// TIA Portal project "智能立库" (V18)

(* hardware
DEVICE "S71500/ET200MP-Station_1"  S7-1500 station
   slot 0: "Profilschiene_0"  Rack  6ES7 590-1***0-0AA0
   slot 0: "PM 70W 120/230VAC"  PM 70W 120/230VAC  6EP1332-4BA00
   slot 1: "PLC_1"  CPU 1516-3 PN/DP  6ES7 516-3AN02-0AB0  V2.9
      slot 3: "CPU-Display_1"  6ES7591-1BA00-0AA0
      slot 32768: "PROFINET-Schnittstelle_1"  X1
         slot 32769: "Port_1"  X1 P1
         slot 32770: "Port_2"  X1 P2
      slot 33024: "PROFINET 接口_1"  X2
      slot 33280: "DP 接口_1"  X3
      slot 34817: "Virtual CP interface port_1"  Virtual CP interface port  Virtual CP interface port
*)

// ===== PLC "PLC_1"  CPU 1516-3 PN/DP =====

VAR_GLOBAL   // PLC tag table "Standard-Variablentabelle"
   "Tag_1" AT %M1000.0 : Bool;
   "Tag_2" AT %M1000.1 : Bool;
   "Tag_3" AT %QW0 : Int;
   "Tag_4" AT %QW1 : Int;
   "Tag_5" AT %QD0 : DWord;
   "Tag_6" AT %QB4 : Byte;
END_VAR

VAR_GLOBAL   // PLC tag table "通讯"
   "确认数量" AT %M200.0 : Bool;
   "出库模式" AT %M200.1 : Bool;
   "入库模式" AT %M200.2 : Bool;
   "启动" AT %M200.3 : Bool;
   "停止" AT %M200.4 : Bool;
   "灰色出库数量" AT %MW202 : Int;
   "绿色出库数量" AT %MW204 : Int;
   "蓝色出库数量" AT %MW206 : Int;
   "取消" AT %M200.5 : Bool;
   "出库启动" AT %M200.6 : Bool;
   "入库启动" AT %M200.7 : Bool;
   "运行标志位" AT %M208.0 : Bool;
   "停止中" AT %M208.1 : Bool;
END_VAR

VAR_GLOBAL   // PLC tag table "仓库数据"
   "1号仓" AT %MW300 : Int;
   "2号仓" AT %MW302 : Int;
   "3号仓" AT %MW304 : Int;
END_VAR

VAR_GLOBAL   // PLC tag table "输入输出"
   "1号仓取货器右移到达" AT %I0.0 : Bool;
   "1号仓取货器左移到达" AT %I0.1 : Bool;
   "1号仓取货器归位" AT %I0.2 : Bool;
   "1号仓取货器运行中" AT %I0.3 : Bool;
   "1号仓码货龙门运行中" AT %I0.4 : Bool;
   "1号仓货物到达传感器" AT %I0.5 : Bool;
   "1号仓货物进入传感器" AT %I0.6 : Bool;
   "1号仓货物离开传感器" AT %I0.7 : Bool;
   "2号仓取货器右移到达" AT %I1.0 : Bool;
   "2号仓取货器左移到达" AT %I1.1 : Bool;
   "2号仓取货器归位" AT %I1.2 : Bool;
   "2号仓取货器运行中" AT %I1.3 : Bool;
   "2号仓码货龙门运行中" AT %I1.4 : Bool;
   "2号仓货物到达传感器" AT %I1.5 : Bool;
   "2号仓货物进入传感器" AT %I1.6 : Bool;
   "2号仓货物离开传感器" AT %I1.7 : Bool;
   "3号仓取货器右移到达" AT %I2.0 : Bool;
   "3号仓取货器左移到达" AT %I2.1 : Bool;
   "3号仓取货器归位" AT %I2.2 : Bool;
   "3号仓取货器运行中" AT %I2.3 : Bool;
   "3号仓码货龙门运行中" AT %I2.4 : Bool;
   "3号仓货物到达传感器" AT %I2.5 : Bool;
   "3号仓货物进入传感器" AT %I2.6 : Bool;
   "3号仓货物离开传感器" AT %I2.7 : Bool;
   "灰色加工中心入料传感器" AT %I3.0 : Bool;
   "灰色加工中心出料传感器" AT %I3.1 : Bool;
   "灰色货箱到达传感器" AT %I3.2 : Bool;
   "绿色加工中心入料传感器" AT %I3.3 : Bool;
   "绿色货箱到达传感器" AT %I3.4 : Bool;
   "绿色加工中心出料传感器" AT %I3.5 : Bool;
   "蓝色加工中心入料传感器" AT %I3.6 : Bool;
   "蓝色加工中心出料传感器" AT %I3.7 : Bool;
   "蓝色货箱到达传感器" AT %I4.0 : Bool;
   "1号仓传送带末端" AT %Q0.0 : Bool;
   "1号仓出货传送带1" AT %Q0.1 : Bool;
   "1号仓出货传送带2" AT %Q0.2 : Bool;
   "1号仓取货器上升" AT %Q0.3 : Bool;
   "1号仓取货器右移" AT %Q0.4 : Bool;
   "1号仓取货器左移" AT %Q0.5 : Bool;
   "1号仓货物进入传送带" AT %Q0.6 : Bool;
   "1号仓进货传送带" AT %Q0.7 : Bool;
   "2号仓传送带末端" AT %Q1.0 : Bool;
   "2号仓出货传送带1" AT %Q1.1 : Bool;
   "2号仓出货传送带2" AT %Q1.2 : Bool;
   "2号仓取货器上升" AT %Q1.3 : Bool;
   "2号仓取货器右移" AT %Q1.4 : Bool;
   "2号仓取货器左移" AT %Q1.5 : Bool;
   "2号仓货物进入传送带" AT %Q1.6 : Bool;
   "2号仓进货传送带" AT %Q1.7 : Bool;
   "3号仓传送带末端" AT %Q2.0 : Bool;
   "3号仓出货传送带1" AT %Q2.1 : Bool;
   "3号仓出货传送带2" AT %Q2.2 : Bool;
   "3号仓取货器上升" AT %Q2.3 : Bool;
   "3号仓取货器右移" AT %Q2.4 : Bool;
   "3号仓取货器左移" AT %Q2.5 : Bool;
   "3号仓货物进入传送带" AT %Q2.6 : Bool;
   "3号仓进货传送带" AT %Q2.7 : Bool;
   "灰色加工中心停止" AT %Q3.0 : Bool;
   "灰色加工中心入料传送带" AT %Q3.1 : Bool;
   "灰色加工中心出料传送带1" AT %Q3.2 : Bool;
   "灰色加工中心出料传送带2" AT %Q3.3 : Bool;
   "灰色加工中心加工上盖使能" AT %Q3.4 : Bool;
   "灰色加工中心启动" AT %Q3.5 : Bool;
   "绿色加工中心停止" AT %Q3.6 : Bool;
   "绿色加工中心入料传送带" AT %Q3.7 : Bool;
   "绿色加工中心出料传送带1" AT %Q4.0 : Bool;
   "绿色加工中心出料传送带2" AT %Q4.1 : Bool;
   "绿色加工中心加工上盖使能" AT %Q4.2 : Bool;
   "绿色加工中心启动" AT %Q4.3 : Bool;
   "蓝色加工中心停止" AT %Q4.4 : Bool;
   "蓝色加工中心入料传送带" AT %Q4.5 : Bool;
   "蓝色加工中心出料传送带1" AT %Q4.6 : Bool;
   "蓝色加工中心出料传送带2" AT %Q4.7 : Bool;
   "蓝色加工中心加工上盖使能" AT %Q5.0 : Bool;
   "蓝色加工中心启动" AT %Q5.1 : Bool;
   "1号仓目标仓位" AT %QD48 : DInt;
   "2号仓目标仓位" AT %QD52 : DInt;
   "3号仓目标仓位" AT %QD56 : DInt;
END_VAR

DATA_BLOCK "模式切换"   // DB1
{ S7_Optimized_Access := 'TRUE' }
VERSION : 0.1
   VAR
      出库模式 : Struct
         中间 : Bool;
         启动 : Bool;
         确认数量 : Bool;
         全部出库完成 : Bool;
      END_STRUCT;
      入库模式 : Struct
         中间 : Bool;
         启动 : Bool;
         入库完成保持 : Struct
            "1" : Bool;
            "2" : Bool;
            "3" : Bool;
            汇总 : Bool;
         END_STRUCT;
      END_STRUCT;
      沿 : Struct
         "1" : Bool;
         "2" : Bool;
         "3" : Bool;
         "4" : Bool;
         "5" : Bool;
      END_STRUCT;
   END_VAR
BEGIN
END_DATA_BLOCK

DATA_BLOCK "2号仓库汇总块_DB"   // DB2
{ S7_Optimized_Access := 'TRUE' }
VERSION : 0.1
// stored: InstanceOfName 汇总块
"汇总块"
BEGIN
END_DATA_BLOCK

DATA_BLOCK "3号仓库汇总块_DB"   // DB3
{ S7_Optimized_Access := 'TRUE' }
VERSION : 0.1
// stored: InstanceOfName 汇总块
"汇总块"
BEGIN
END_DATA_BLOCK

DATA_BLOCK "手动调试模式数据"   // DB4
{ S7_Optimized_Access := 'FALSE' }
VERSION : 0.1
   VAR
      传感器数据 : Struct
         "1号仓取货器右移到达" : Bool;
         "1号仓取货器左移到达" : Bool;
         "1号仓取货器归位" : Bool;
         "1号仓取货器运行中" : Bool;
         "1号仓码货龙门运行中" : Bool;
         "1号仓货物到达传感器" : Bool;
         "1号仓货物进入传感器" : Bool;
         "1号仓货物离开传感器" : Bool;
         "2号仓取货器右移到达" : Bool;
         "2号仓取货器左移到达" : Bool;
         "2号仓取货器归位" : Bool;
         "2号仓取货器运行中" : Bool;
         "2号仓码货龙门运行中" : Bool;
         "2号仓货物到达传感器" : Bool;
         "2号仓货物进入传感器" : Bool;
         "2号仓货物离开传感器" : Bool;
         "3号仓取货器右移到达" : Bool;
         "3号仓取货器左移到达" : Bool;
         "3号仓取货器归位" : Bool;
         "3号仓取货器运行中" : Bool;
         "3号仓码货龙门运行中" : Bool;
         "3号仓货物到达传感器" : Bool;
         "3号仓货物进入传感器" : Bool;
         "3号仓货物离开传感器" : Bool;
         灰色加工中心入料传感器 : Bool;
         灰色加工中心出料传感器 : Bool;
         灰色货箱到达传感器 : Bool;
         绿色加工中心入料传感器 : Bool;
         绿色货箱到达传感器 : Bool;
         绿色加工中心出料传感器 : Bool;
         蓝色加工中心入料传感器 : Bool;
         蓝色加工中心出料传感器 : Bool;
         蓝色货箱到达传感器 : Bool;
      END_STRUCT;
      执行器 : Struct
         "1号仓传送带末端" : Bool;
         "1号仓出货传送带1" : Bool;
         "1号仓出货传送带2" : Bool;
         "1号仓取货器上升" : Bool;
         "1号仓取货器右移" : Bool;
         "1号仓取货器左移" : Bool;
         "1号仓货物进入传送带" : Bool;
         "1号仓进货传送带" : Bool;
         "2号仓传送带末端" : Bool;
         "2号仓出货传送带1" : Bool;
         "2号仓出货传送带2" : Bool;
         "2号仓取货器上升" : Bool;
         "2号仓取货器右移" : Bool;
         "2号仓取货器左移" : Bool;
         "2号仓货物进入传送带" : Bool;
         "2号仓进货传送带" : Bool;
         "3号仓传送带末端" : Bool;
         "3号仓出货传送带1" : Bool;
         "3号仓出货传送带2" : Bool;
         "3号仓取货器上升" : Bool;
         "3号仓取货器右移" : Bool;
         "3号仓取货器左移" : Bool;
         "3号仓货物进入传送带" : Bool;
         "3号仓进货传送带" : Bool;
         灰色加工中心停止 : Bool;
         灰色加工中心入料传送带 : Bool;
         灰色加工中心出料传送带1 : Bool;
         灰色加工中心出料传送带2 : Bool;
         灰色加工中心加工上盖使能 : Bool;
         灰色加工中心启动 : Bool;
         绿色加工中心停止 : Bool;
         绿色加工中心入料传送带 : Bool;
         绿色加工中心出料传送带1 : Bool;
         绿色加工中心出料传送带2 : Bool;
         绿色加工中心加工上盖使能 : Bool;
         绿色加工中心启动 : Bool;
         蓝色加工中心停止 : Bool;
         蓝色加工中心入料传送带 : Bool;
         蓝色加工中心出料传送带1 : Bool;
         蓝色加工中心出料传送带2 : Bool;
         蓝色加工中心加工上盖使能 : Bool;
         蓝色加工中心启动 : Bool;
      END_STRUCT;
   END_VAR
BEGIN
END_DATA_BLOCK

DATA_BLOCK "1号仓库汇总块_DB"   // DB7
{ S7_Optimized_Access := 'TRUE' }
VERSION : 0.1
// stored: InstanceOfName 汇总块
"汇总块"
BEGIN
END_DATA_BLOCK

FUNCTION_BLOCK "取货器"   // FB1, LAD
{ S7_Optimized_Access := 'TRUE' }
VERSION : 0.1
   VAR_INPUT
      传送带进货 : Bool;
      "传送带出货/仓库进货" : Bool;
      仓库出货 : Bool;
      取货器左移到达 : Bool;
      取货器右移到达 : Bool;
      取货器归位 : Bool;
      取货器运行中 : Bool;
   END_VAR
   VAR_OUTPUT
      取货臂左移 : Bool;
      取货臂右移 : Bool;
      取货器上升 : Bool;
      传送带进货完成 : Bool;
      "传送带出货/仓库进货完成" : Bool;
      仓库出货完成 : Bool;
   END_VAR
   VAR
      传送带进货运行步 : Int;
      传送带出货运行步 : Int;
      仓库出货运行步 : Int;
      传送带进货沿缓冲位 : Struct
         "1" : Bool;
         "2" : Bool;
         "3" : Bool;
         "4" : Bool;
         "5" : Bool;
         "6" : Bool;
      END_STRUCT;
      "传送带出货/仓库进货沿缓冲位" : Struct
         "1" : Bool;
         "2" : Bool;
         "3" : Bool;
         "4" : Bool;
         "5" : Bool;
      END_STRUCT;
      仓库出货沿缓冲位 : Struct
         "1" : Bool;
         "2" : Bool;
         "3" : Bool;
         "4" : Bool;
         "5" : Bool;
      END_STRUCT;
   END_VAR
   VAR_TEMP   // added for the SCL form of the ladder/FBD networks
      _w1 : Bool;
      _w2 : Bool;
      _w3 : Bool;
      _w4 : Bool;
      _w5 : Bool;
      _w6 : Bool;
      _w7 : Bool;
      _w8 : Bool;
      _w9 : Bool;
   END_VAR
BEGIN

REGION Network 1: 传送带进货
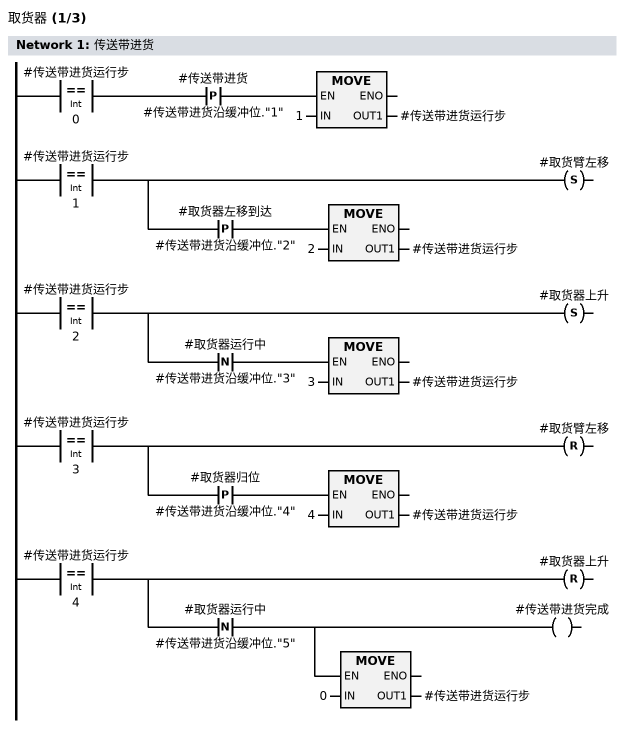
   RUNG wire#powerrail
      { S7_Templates := "SrcType := Int" } EQ_Contact(in1 := #传送带进货运行步, in2 := 0)
      P_Contact(operand := #传送带进货, bit := #传送带进货沿缓冲位."1")
      Move(in := 1, out1 => #传送带进货运行步)
   END_RUNG
   RUNG wire#powerrail
      { S7_Templates := "SrcType := Int" } EQ_Contact(in1 := #传送带进货运行步, in2 := 1)
      wire#w1
      S_Coil( #取货臂左移 )
   END_RUNG
   RUNG wire#w1
      P_Contact(operand := #取货器左移到达, bit := #传送带进货沿缓冲位."2")
      Move(in := 2, out1 => #传送带进货运行步)
   END_RUNG
   RUNG wire#powerrail
      { S7_Templates := "SrcType := Int" } EQ_Contact(in1 := #传送带进货运行步, in2 := 2)
      wire#w2
      S_Coil( #取货器上升 )
   END_RUNG
   RUNG wire#w2
      N_Contact(operand := #取货器运行中, bit := #传送带进货沿缓冲位."3")
      Move(in := 3, out1 => #传送带进货运行步)
   END_RUNG
   RUNG wire#powerrail
      { S7_Templates := "SrcType := Int" } EQ_Contact(in1 := #传送带进货运行步, in2 := 3)
      wire#w3
      R_Coil( #取货臂左移 )
   END_RUNG
   RUNG wire#w3
      P_Contact(operand := #取货器归位, bit := #传送带进货沿缓冲位."4")
      Move(in := 4, out1 => #传送带进货运行步)
   END_RUNG
   RUNG wire#powerrail
      { S7_Templates := "SrcType := Int" } EQ_Contact(in1 := #传送带进货运行步, in2 := 4)
      wire#w4
      R_Coil( #取货器上升 )
   END_RUNG
   RUNG wire#w4
      N_Contact(operand := #取货器运行中, bit := #传送带进货沿缓冲位."5")
      wire#w5
      Coil( #传送带进货完成 )
   END_RUNG
   RUNG wire#w5
      Move(in := 0, out1 => #传送带进货运行步)
   END_RUNG
   // the same network as SCL:
   #_w1 := (#传送带进货运行步 = 0) AND #传送带进货 AND NOT #传送带进货沿缓冲位."1";   // rising edge of #传送带进货
   #传送带进货沿缓冲位."1" := #传送带进货;
   IF #_w1 THEN #传送带进货运行步 := 1; END_IF;
   #_w2 := #传送带进货运行步 = 1;
   IF #_w2 THEN #取货臂左移 := TRUE; END_IF;
   #_w3 := #_w2 AND #取货器左移到达 AND NOT #传送带进货沿缓冲位."2";   // rising edge of #取货器左移到达
   #传送带进货沿缓冲位."2" := #取货器左移到达;
   IF #_w3 THEN #传送带进货运行步 := 2; END_IF;
   #_w4 := #传送带进货运行步 = 2;
   IF #_w4 THEN #取货器上升 := TRUE; END_IF;
   #_w5 := #_w4 AND NOT #取货器运行中 AND #传送带进货沿缓冲位."3";   // falling edge of #取货器运行中
   #传送带进货沿缓冲位."3" := #取货器运行中;
   IF #_w5 THEN #传送带进货运行步 := 3; END_IF;
   #_w6 := #传送带进货运行步 = 3;
   IF #_w6 THEN #取货臂左移 := FALSE; END_IF;
   #_w7 := #_w6 AND #取货器归位 AND NOT #传送带进货沿缓冲位."4";   // rising edge of #取货器归位
   #传送带进货沿缓冲位."4" := #取货器归位;
   IF #_w7 THEN #传送带进货运行步 := 4; END_IF;
   #_w8 := #传送带进货运行步 = 4;
   IF #_w8 THEN #取货器上升 := FALSE; END_IF;
   #_w9 := #_w8 AND NOT #取货器运行中 AND #传送带进货沿缓冲位."5";   // falling edge of #取货器运行中
   #传送带进货沿缓冲位."5" := #取货器运行中;
   #传送带进货完成 := #_w9;
   IF #_w9 THEN #传送带进货运行步 := 0; END_IF;
END_REGION

REGION Network 2: 传送带出货/仓库进货
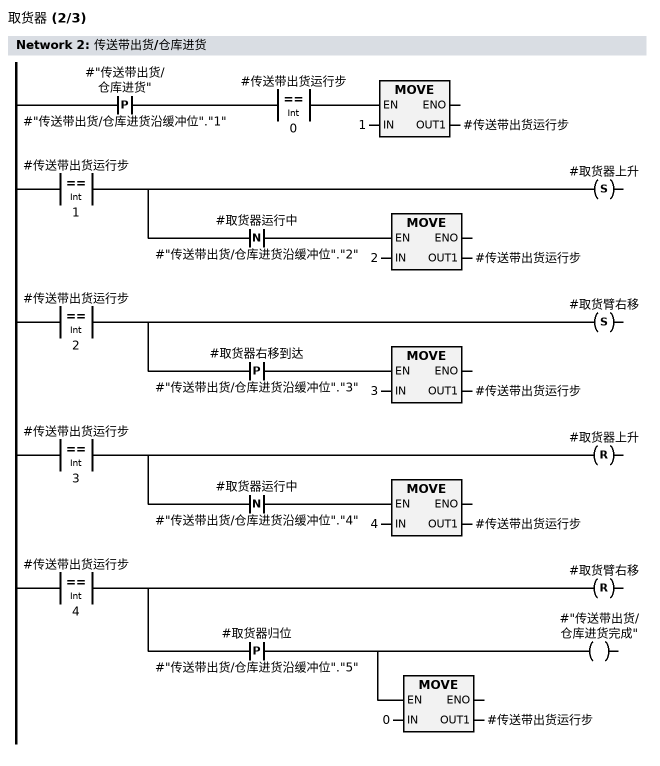
   RUNG wire#powerrail
      P_Contact(operand := #"传送带出货/仓库进货", bit := #"传送带出货/仓库进货沿缓冲位"."1")
      { S7_Templates := "SrcType := Int" } EQ_Contact(in1 := #传送带出货运行步, in2 := 0)
      Move(in := 1, out1 => #传送带出货运行步)
   END_RUNG
   RUNG wire#powerrail
      { S7_Templates := "SrcType := Int" } EQ_Contact(in1 := #传送带出货运行步, in2 := 1)
      wire#w1
      S_Coil( #取货器上升 )
   END_RUNG
   RUNG wire#w1
      N_Contact(operand := #取货器运行中, bit := #"传送带出货/仓库进货沿缓冲位"."2")
      Move(in := 2, out1 => #传送带出货运行步)
   END_RUNG
   RUNG wire#powerrail
      { S7_Templates := "SrcType := Int" } EQ_Contact(in1 := #传送带出货运行步, in2 := 2)
      wire#w2
      S_Coil( #取货臂右移 )
   END_RUNG
   RUNG wire#w2
      P_Contact(operand := #取货器右移到达, bit := #"传送带出货/仓库进货沿缓冲位"."3")
      Move(in := 3, out1 => #传送带出货运行步)
   END_RUNG
   RUNG wire#powerrail
      { S7_Templates := "SrcType := Int" } EQ_Contact(in1 := #传送带出货运行步, in2 := 3)
      wire#w3
      R_Coil( #取货器上升 )
   END_RUNG
   RUNG wire#w3
      N_Contact(operand := #取货器运行中, bit := #"传送带出货/仓库进货沿缓冲位"."4")
      Move(in := 4, out1 => #传送带出货运行步)
   END_RUNG
   RUNG wire#powerrail
      { S7_Templates := "SrcType := Int" } EQ_Contact(in1 := #传送带出货运行步, in2 := 4)
      wire#w4
      R_Coil( #取货臂右移 )
   END_RUNG
   RUNG wire#w4
      P_Contact(operand := #取货器归位, bit := #"传送带出货/仓库进货沿缓冲位"."5")
      wire#w5
      Coil( #"传送带出货/仓库进货完成" )
   END_RUNG
   RUNG wire#w5
      Move(in := 0, out1 => #传送带出货运行步)
   END_RUNG
   // the same network as SCL:
   #_w1 := #"传送带出货/仓库进货" AND NOT #"传送带出货/仓库进货沿缓冲位"."1";   // rising edge of #"传送带出货/仓库进货"
   #"传送带出货/仓库进货沿缓冲位"."1" := #"传送带出货/仓库进货";
   IF #_w1 AND (#传送带出货运行步 = 0) THEN #传送带出货运行步 := 1; END_IF;
   #_w2 := #传送带出货运行步 = 1;
   IF #_w2 THEN #取货器上升 := TRUE; END_IF;
   #_w3 := #_w2 AND NOT #取货器运行中 AND #"传送带出货/仓库进货沿缓冲位"."2";   // falling edge of #取货器运行中
   #"传送带出货/仓库进货沿缓冲位"."2" := #取货器运行中;
   IF #_w3 THEN #传送带出货运行步 := 2; END_IF;
   #_w4 := #传送带出货运行步 = 2;
   IF #_w4 THEN #取货臂右移 := TRUE; END_IF;
   #_w5 := #_w4 AND #取货器右移到达 AND NOT #"传送带出货/仓库进货沿缓冲位"."3";   // rising edge of #取货器右移到达
   #"传送带出货/仓库进货沿缓冲位"."3" := #取货器右移到达;
   IF #_w5 THEN #传送带出货运行步 := 3; END_IF;
   #_w6 := #传送带出货运行步 = 3;
   IF #_w6 THEN #取货器上升 := FALSE; END_IF;
   #_w7 := #_w6 AND NOT #取货器运行中 AND #"传送带出货/仓库进货沿缓冲位"."4";   // falling edge of #取货器运行中
   #"传送带出货/仓库进货沿缓冲位"."4" := #取货器运行中;
   IF #_w7 THEN #传送带出货运行步 := 4; END_IF;
   #_w8 := #传送带出货运行步 = 4;
   IF #_w8 THEN #取货臂右移 := FALSE; END_IF;
   #_w9 := #_w8 AND #取货器归位 AND NOT #"传送带出货/仓库进货沿缓冲位"."5";   // rising edge of #取货器归位
   #"传送带出货/仓库进货沿缓冲位"."5" := #取货器归位;
   #"传送带出货/仓库进货完成" := #_w9;
   IF #_w9 THEN #传送带出货运行步 := 0; END_IF;
END_REGION

REGION Network 3: 仓库出货
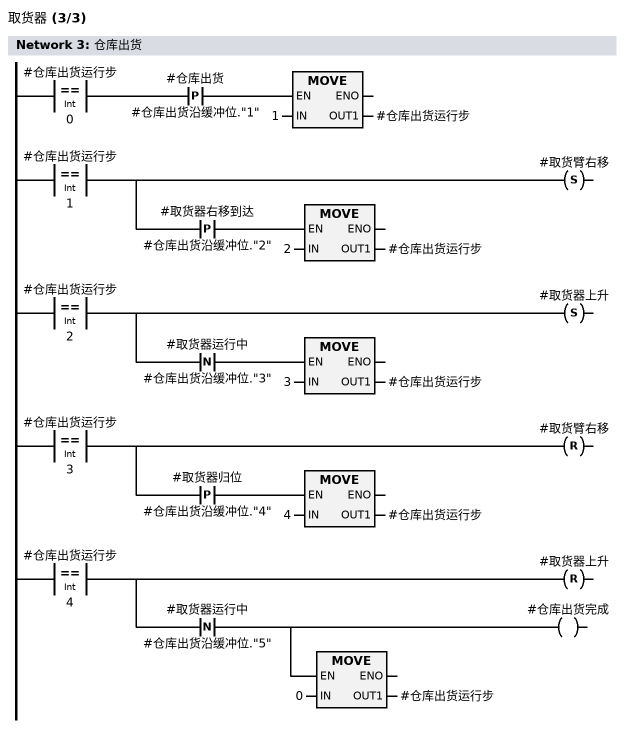
   RUNG wire#powerrail
      { S7_Templates := "SrcType := Int" } EQ_Contact(in1 := #仓库出货运行步, in2 := 0)
      P_Contact(operand := #仓库出货, bit := #仓库出货沿缓冲位."1")
      Move(in := 1, out1 => #仓库出货运行步)
   END_RUNG
   RUNG wire#powerrail
      { S7_Templates := "SrcType := Int" } EQ_Contact(in1 := #仓库出货运行步, in2 := 1)
      wire#w1
      S_Coil( #取货臂右移 )
   END_RUNG
   RUNG wire#w1
      P_Contact(operand := #取货器右移到达, bit := #仓库出货沿缓冲位."2")
      Move(in := 2, out1 => #仓库出货运行步)
   END_RUNG
   RUNG wire#powerrail
      { S7_Templates := "SrcType := Int" } EQ_Contact(in1 := #仓库出货运行步, in2 := 2)
      wire#w2
      S_Coil( #取货器上升 )
   END_RUNG
   RUNG wire#w2
      N_Contact(operand := #取货器运行中, bit := #仓库出货沿缓冲位."3")
      Move(in := 3, out1 => #仓库出货运行步)
   END_RUNG
   RUNG wire#powerrail
      { S7_Templates := "SrcType := Int" } EQ_Contact(in1 := #仓库出货运行步, in2 := 3)
      wire#w3
      R_Coil( #取货臂右移 )
   END_RUNG
   RUNG wire#w3
      P_Contact(operand := #取货器归位, bit := #仓库出货沿缓冲位."4")
      Move(in := 4, out1 => #仓库出货运行步)
   END_RUNG
   RUNG wire#powerrail
      { S7_Templates := "SrcType := Int" } EQ_Contact(in1 := #仓库出货运行步, in2 := 4)
      wire#w4
      R_Coil( #取货器上升 )
   END_RUNG
   RUNG wire#w4
      N_Contact(operand := #取货器运行中, bit := #仓库出货沿缓冲位."5")
      wire#w5
      Coil( #仓库出货完成 )
   END_RUNG
   RUNG wire#w5
      Move(in := 0, out1 => #仓库出货运行步)
   END_RUNG
   // the same network as SCL:
   #_w1 := (#仓库出货运行步 = 0) AND #仓库出货 AND NOT #仓库出货沿缓冲位."1";   // rising edge of #仓库出货
   #仓库出货沿缓冲位."1" := #仓库出货;
   IF #_w1 THEN #仓库出货运行步 := 1; END_IF;
   #_w2 := #仓库出货运行步 = 1;
   IF #_w2 THEN #取货臂右移 := TRUE; END_IF;
   #_w3 := #_w2 AND #取货器右移到达 AND NOT #仓库出货沿缓冲位."2";   // rising edge of #取货器右移到达
   #仓库出货沿缓冲位."2" := #取货器右移到达;
   IF #_w3 THEN #仓库出货运行步 := 2; END_IF;
   #_w4 := #仓库出货运行步 = 2;
   IF #_w4 THEN #取货器上升 := TRUE; END_IF;
   #_w5 := #_w4 AND NOT #取货器运行中 AND #仓库出货沿缓冲位."3";   // falling edge of #取货器运行中
   #仓库出货沿缓冲位."3" := #取货器运行中;
   IF #_w5 THEN #仓库出货运行步 := 3; END_IF;
   #_w6 := #仓库出货运行步 = 3;
   IF #_w6 THEN #取货臂右移 := FALSE; END_IF;
   #_w7 := #_w6 AND #取货器归位 AND NOT #仓库出货沿缓冲位."4";   // rising edge of #取货器归位
   #仓库出货沿缓冲位."4" := #取货器归位;
   IF #_w7 THEN #仓库出货运行步 := 4; END_IF;
   #_w8 := #仓库出货运行步 = 4;
   IF #_w8 THEN #取货器上升 := FALSE; END_IF;
   #_w9 := #_w8 AND NOT #取货器运行中 AND #仓库出货沿缓冲位."5";   // falling edge of #取货器运行中
   #仓库出货沿缓冲位."5" := #取货器运行中;
   #仓库出货完成 := #_w9;
   IF #_w9 THEN #仓库出货运行步 := 0; END_IF;
END_REGION
END_FUNCTION_BLOCK

FUNCTION_BLOCK "龙门码货机"   // FB2, LAD
{ S7_Optimized_Access := 'TRUE' }
VERSION : 0.1
   VAR_INPUT
      仓位号输入 : Int;
      入库 : Bool;
      出库 : Bool;
      龙门运行中 : Bool;
      取货器左移到达传感器 : Bool;
      取货器右移到达传感器 : Bool;
      取货器归位传感器 : Bool;
      取货器运行传感器 : Bool;
   END_VAR
   VAR_OUTPUT
      仓位号输出 : DInt;
      取货臂左移 : Bool;
      取货臂右移 : Bool;
      取货器上升 : Bool;
      入库完成 : Bool;
      出库完成 : Bool;
   END_VAR
   VAR
      入库步骤号 : Int;
      出库步骤号 : Int;
      入库沿缓冲位 : Struct
         "1" : Bool;
         "2" : Bool;
         "3" : Bool;
         "4" : Bool;
      END_STRUCT;
      出库沿缓冲位 : Struct
         "1" : Bool;
         "2" : Bool;
         "3" : Bool;
         "4" : Bool;
      END_STRUCT;
      取货器_Instance : "取货器";
   END_VAR
   VAR_TEMP   // added for the SCL form of the ladder/FBD networks
      _w1 : Bool;
      _w2 : Bool;
      _w3 : Bool;
      _w4 : Bool;
      _w5 : Bool;
      _w6 : Bool;
      _w7 : Bool;
      _w8 : Bool;
      _w9 : Bool;
   END_VAR
BEGIN

REGION Network 1: 入库
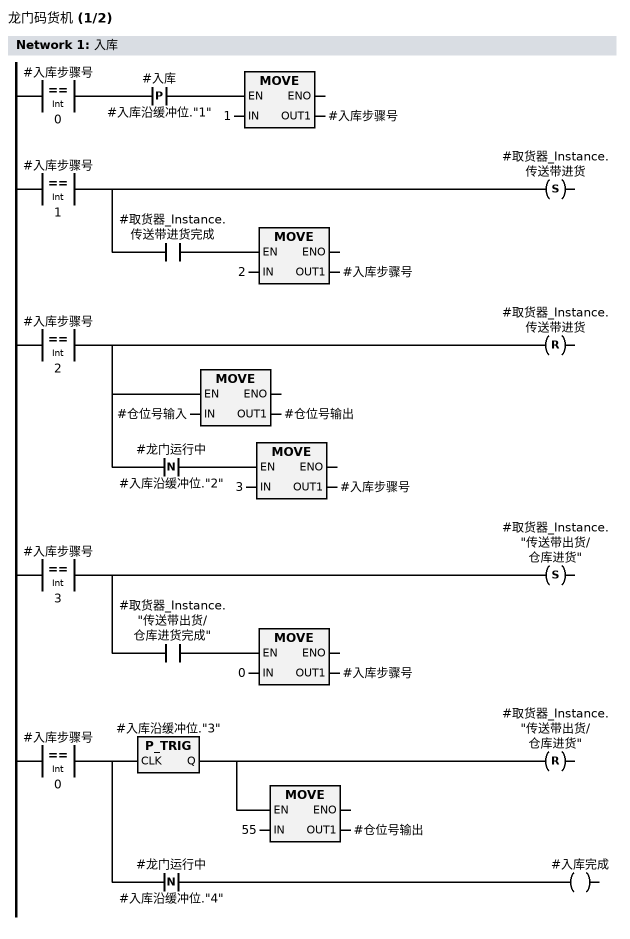
   RUNG wire#powerrail
      { S7_Templates := "SrcType := Int" } EQ_Contact(in1 := #入库步骤号, in2 := 0)
      P_Contact(operand := #入库, bit := #入库沿缓冲位."1")
      Move(in := 1, out1 => #入库步骤号)
   END_RUNG
   RUNG wire#powerrail
      { S7_Templates := "SrcType := Int" } EQ_Contact(in1 := #入库步骤号, in2 := 1)
      wire#w1
      S_Coil( #取货器_Instance.传送带进货 )
   END_RUNG
   RUNG wire#w1
      Contact( #取货器_Instance.传送带进货完成 )
      Move(in := 2, out1 => #入库步骤号)
   END_RUNG
   RUNG wire#powerrail
      { S7_Templates := "SrcType := Int" } EQ_Contact(in1 := #入库步骤号, in2 := 2)
      wire#w2
      R_Coil( #取货器_Instance.传送带进货 )
   END_RUNG
   RUNG wire#w2
      Move(in := #仓位号输入, out1 => #仓位号输出)
   END_RUNG
   RUNG wire#w2
      N_Contact(operand := #龙门运行中, bit := #入库沿缓冲位."2")
      Move(in := 3, out1 => #入库步骤号)
   END_RUNG
   RUNG wire#powerrail
      { S7_Templates := "SrcType := Int" } EQ_Contact(in1 := #入库步骤号, in2 := 3)
      wire#w3
      S_Coil( #取货器_Instance."传送带出货/仓库进货" )
   END_RUNG
   RUNG wire#w3
      Contact( #取货器_Instance."传送带出货/仓库进货完成" )
      Move(in := 0, out1 => #入库步骤号)
   END_RUNG
   RUNG wire#powerrail
      { S7_Templates := "SrcType := Int" } EQ_Contact(in1 := #入库步骤号, in2 := 0)
      wire#w4
      P_Trig( #入库沿缓冲位."3" )
      wire#w5
      R_Coil( #取货器_Instance."传送带出货/仓库进货" )
   END_RUNG
   RUNG wire#w5
      Move(in := 55, out1 => #仓位号输出)
   END_RUNG
   RUNG wire#w4
      N_Contact(operand := #龙门运行中, bit := #入库沿缓冲位."4")
      Coil( #入库完成 )
   END_RUNG
   // the same network as SCL:
   #_w1 := (#入库步骤号 = 0) AND #入库 AND NOT #入库沿缓冲位."1";   // rising edge of #入库
   #入库沿缓冲位."1" := #入库;
   IF #_w1 THEN #入库步骤号 := 1; END_IF;
   #_w2 := #入库步骤号 = 1;
   IF #_w2 THEN #取货器_Instance.传送带进货 := TRUE; END_IF;
   IF #_w2 AND #取货器_Instance.传送带进货完成 THEN #入库步骤号 := 2; END_IF;
   #_w3 := #入库步骤号 = 2;
   IF #_w3 THEN
       #取货器_Instance.传送带进货 := FALSE;
       #仓位号输出 := #仓位号输入;
   END_IF;
   #_w4 := #_w3 AND NOT #龙门运行中 AND #入库沿缓冲位."2";   // falling edge of #龙门运行中
   #入库沿缓冲位."2" := #龙门运行中;
   IF #_w4 THEN #入库步骤号 := 3; END_IF;
   #_w5 := #入库步骤号 = 3;
   IF #_w5 THEN #取货器_Instance."传送带出货/仓库进货" := TRUE; END_IF;
   IF #_w5 AND #取货器_Instance."传送带出货/仓库进货完成" THEN #入库步骤号 := 0; END_IF;
   #_w6 := #入库步骤号 = 0;
   #_w7 := #_w6 AND NOT #入库沿缓冲位."3";   // rising edge
   #入库沿缓冲位."3" := #_w6;
   IF #_w7 THEN
       #取货器_Instance."传送带出货/仓库进货" := FALSE;
       #仓位号输出 := 55;
   END_IF;
   #_w8 := #_w6 AND NOT #龙门运行中 AND #入库沿缓冲位."4";   // falling edge of #龙门运行中
   #入库沿缓冲位."4" := #龙门运行中;
   #入库完成 := #_w8;
END_REGION

REGION Network 2: 出库
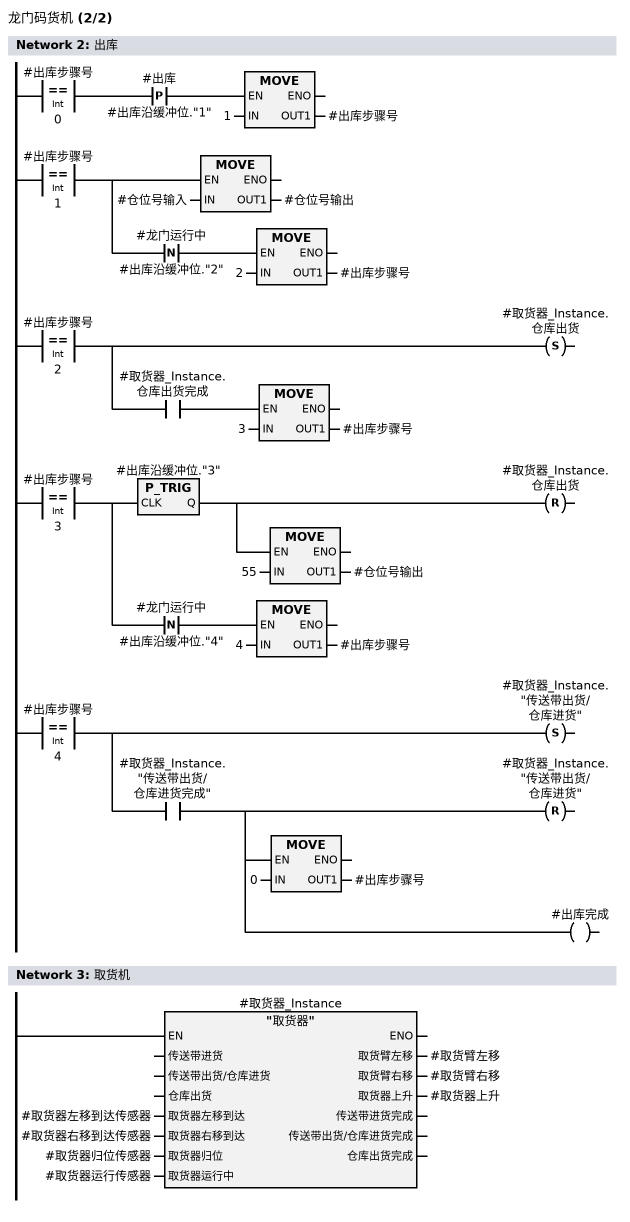
   RUNG wire#powerrail
      { S7_Templates := "SrcType := Int" } EQ_Contact(in1 := #出库步骤号, in2 := 0)
      P_Contact(operand := #出库, bit := #出库沿缓冲位."1")
      Move(in := 1, out1 => #出库步骤号)
   END_RUNG
   RUNG wire#powerrail
      { S7_Templates := "SrcType := Int" } EQ_Contact(in1 := #出库步骤号, in2 := 1)
      wire#w1
      Move(in := #仓位号输入, out1 => #仓位号输出)
   END_RUNG
   RUNG wire#w1
      N_Contact(operand := #龙门运行中, bit := #出库沿缓冲位."2")
      Move(in := 2, out1 => #出库步骤号)
   END_RUNG
   RUNG wire#powerrail
      { S7_Templates := "SrcType := Int" } EQ_Contact(in1 := #出库步骤号, in2 := 2)
      wire#w2
      S_Coil( #取货器_Instance.仓库出货 )
   END_RUNG
   RUNG wire#w2
      Contact( #取货器_Instance.仓库出货完成 )
      Move(in := 3, out1 => #出库步骤号)
   END_RUNG
   RUNG wire#powerrail
      { S7_Templates := "SrcType := Int" } EQ_Contact(in1 := #出库步骤号, in2 := 3)
      wire#w3
      P_Trig( #出库沿缓冲位."3" )
      wire#w4
      R_Coil( #取货器_Instance.仓库出货 )
   END_RUNG
   RUNG wire#w4
      Move(in := 55, out1 => #仓位号输出)
   END_RUNG
   RUNG wire#w3
      N_Contact(operand := #龙门运行中, bit := #出库沿缓冲位."4")
      Move(in := 4, out1 => #出库步骤号)
   END_RUNG
   RUNG wire#powerrail
      { S7_Templates := "SrcType := Int" } EQ_Contact(in1 := #出库步骤号, in2 := 4)
      wire#w5
      S_Coil( #取货器_Instance."传送带出货/仓库进货" )
   END_RUNG
   RUNG wire#w5
      Contact( #取货器_Instance."传送带出货/仓库进货完成" )
      wire#w6
      R_Coil( #取货器_Instance."传送带出货/仓库进货" )
   END_RUNG
   RUNG wire#w6
      Move(in := 0, out1 => #出库步骤号)
   END_RUNG
   RUNG wire#w6
      Coil( #出库完成 )
   END_RUNG
   // the same network as SCL:
   #_w1 := (#出库步骤号 = 0) AND #出库 AND NOT #出库沿缓冲位."1";   // rising edge of #出库
   #出库沿缓冲位."1" := #出库;
   IF #_w1 THEN #出库步骤号 := 1; END_IF;
   #_w2 := #出库步骤号 = 1;
   IF #_w2 THEN #仓位号输出 := #仓位号输入; END_IF;
   #_w3 := #_w2 AND NOT #龙门运行中 AND #出库沿缓冲位."2";   // falling edge of #龙门运行中
   #出库沿缓冲位."2" := #龙门运行中;
   IF #_w3 THEN #出库步骤号 := 2; END_IF;
   #_w4 := #出库步骤号 = 2;
   IF #_w4 THEN #取货器_Instance.仓库出货 := TRUE; END_IF;
   IF #_w4 AND #取货器_Instance.仓库出货完成 THEN #出库步骤号 := 3; END_IF;
   #_w5 := #出库步骤号 = 3;
   #_w6 := #_w5 AND NOT #出库沿缓冲位."3";   // rising edge
   #出库沿缓冲位."3" := #_w5;
   IF #_w6 THEN
       #取货器_Instance.仓库出货 := FALSE;
       #仓位号输出 := 55;
   END_IF;
   #_w7 := #_w5 AND NOT #龙门运行中 AND #出库沿缓冲位."4";   // falling edge of #龙门运行中
   #出库沿缓冲位."4" := #龙门运行中;
   IF #_w7 THEN #出库步骤号 := 4; END_IF;
   #_w8 := #出库步骤号 = 4;
   IF #_w8 THEN #取货器_Instance."传送带出货/仓库进货" := TRUE; END_IF;
   #_w9 := #_w8 AND #取货器_Instance."传送带出货/仓库进货完成";
   IF #_w9 THEN
       #取货器_Instance."传送带出货/仓库进货" := FALSE;
       #出库步骤号 := 0;
   END_IF;
   #出库完成 := #_w9;
END_REGION

REGION Network 3: 取货机
   RUNG wire#powerrail
      #取货器_Instance(传送带进货 :=, "传送带出货/仓库进货" :=, 仓库出货 :=, 取货器左移到达 := #取货器左移到达传感器, 取货器右移到达 := #取货器右移到达传感器, 取货器归位 := #取货器归位传感器, 取货器运行中 := #取货器运行传感器, 取货臂左移 => #取货臂左移, 取货臂右移 => #取货臂右移, 取货器上升 => #取货器上升, 传送带进货完成 =>, "传送带出货/仓库进货完成" =>, 仓库出货完成 =>)
   END_RUNG
   // the same network as SCL:
   #取货器_Instance(取货器左移到达 := #取货器左移到达传感器,   // "取货器"
                 取货器右移到达 := #取货器右移到达传感器,
                 取货器归位 := #取货器归位传感器,
                 取货器运行中 := #取货器运行传感器,
                 取货臂左移 => #取货臂左移,
                 取货臂右移 => #取货臂右移,
                 取货器上升 => #取货器上升);
END_REGION
END_FUNCTION_BLOCK

FUNCTION_BLOCK "进出库调度"   // FB3, LAD
{ S7_Optimized_Access := 'TRUE' }
VERSION : 0.1
   VAR_INPUT
      出库模式 : Bool;
      入库模式 : Bool;
      入库完成 : Bool;
      出库完成 : Bool;
      货物到达 : Bool;
      货物进入 : Bool;
      货物离开 : Bool;
      出库数量 : Int;
      确认数量 : Bool;
   END_VAR
   VAR_OUTPUT
      仓库位号输出 : Int;
      启动入库 : Bool;
      启动出库 : Bool;
      完成出库或未启动出库 : Bool;
      满仓 : Bool;
      无货 : Bool;
      入库模式暂存位 : Bool;
      加工中心加工中 : Bool;
   END_VAR
   VAR_IN_OUT
      仓库货物数量 : Int;
   END_VAR
   VAR
      货物到达_沿缓冲位 : Struct
         "1" : Bool;
         "2" : Bool;
      END_STRUCT;
      货物离开_沿缓冲位 : Struct
         "1" : Bool;
         "2" : Bool;
      END_STRUCT;
      运行标志位 : Struct
         出库运行中 : Bool;
         入库运行中 : Bool;
      END_STRUCT;
      取出数量暂存 : Int;
      启动出库暂存 : Struct
         "1" : Bool;
         "2" : Bool;
      END_STRUCT;
   END_VAR
   VAR_TEMP   // added for the SCL form of the ladder/FBD networks
      _w1 : Bool;
      _w2 : Bool;
   END_VAR
BEGIN

REGION Network 1: 入库操作
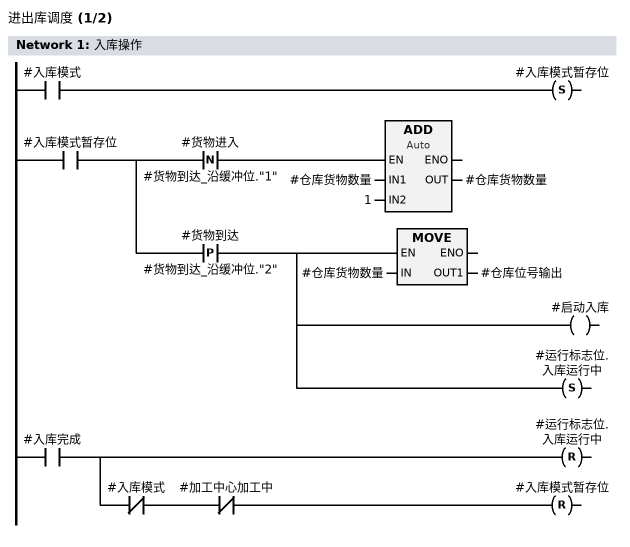
   RUNG wire#powerrail
      Contact( #入库模式 )
      S_Coil( #入库模式暂存位 )
   END_RUNG
   RUNG wire#powerrail
      Contact( #入库模式暂存位 )
      wire#w1
      N_Contact(operand := #货物进入, bit := #货物到达_沿缓冲位."1")
      Add(in1 := #仓库货物数量, in2 := 1, out => #仓库货物数量)
   END_RUNG
   RUNG wire#w1
      P_Contact(operand := #货物到达, bit := #货物到达_沿缓冲位."2")
      wire#w2
      Move(in := #仓库货物数量, out1 => #仓库位号输出)
   END_RUNG
   RUNG wire#w2
      Coil( #启动入库 )
   END_RUNG
   RUNG wire#w2
      S_Coil( #运行标志位.入库运行中 )
   END_RUNG
   RUNG wire#powerrail
      Contact( #入库完成 )
      wire#w3
      R_Coil( #运行标志位.入库运行中 )
   END_RUNG
   RUNG wire#w3
      I_Contact( #入库模式 )
      I_Contact( #加工中心加工中 )
      R_Coil( #入库模式暂存位 )
   END_RUNG
   // the same network as SCL:
   IF #入库模式 THEN #入库模式暂存位 := TRUE; END_IF;
   #_w1 := #入库模式暂存位 AND NOT #货物进入 AND #货物到达_沿缓冲位."1";   // falling edge of #货物进入
   #货物到达_沿缓冲位."1" := #货物进入;
   IF #_w1 THEN #仓库货物数量 := #仓库货物数量 + 1; END_IF;
   #_w2 := #入库模式暂存位 AND #货物到达 AND NOT #货物到达_沿缓冲位."2";   // rising edge of #货物到达
   #货物到达_沿缓冲位."2" := #货物到达;
   IF #_w2 THEN #仓库位号输出 := #仓库货物数量; END_IF;
   #启动入库 := #_w2;
   IF #_w2 THEN #运行标志位.入库运行中 := TRUE; END_IF;
   IF #入库完成 THEN #运行标志位.入库运行中 := FALSE; END_IF;
   IF #入库完成 AND NOT #入库模式 AND NOT #加工中心加工中 THEN #入库模式暂存位 := FALSE; END_IF;
END_REGION

REGION Network 2: 出库操作
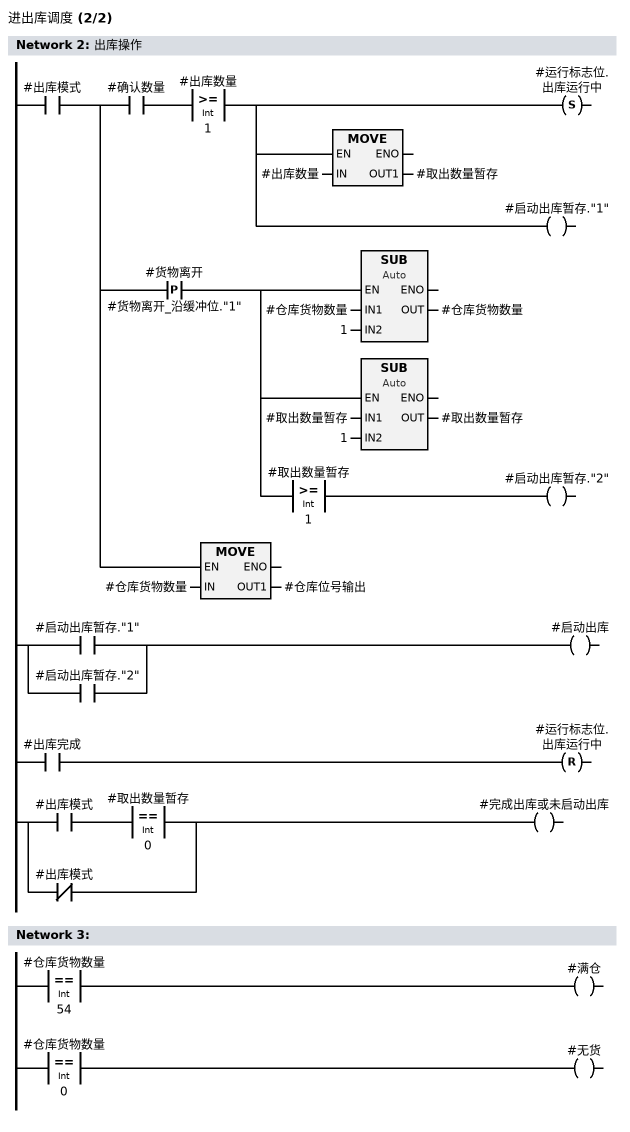
   RUNG wire#powerrail
      Contact( #出库模式 )
      wire#w1
      Contact( #确认数量 )
      { S7_Templates := "SrcType := Int" } GE_Contact(in1 := #出库数量, in2 := 1)
      wire#w2
      S_Coil( #运行标志位.出库运行中 )
   END_RUNG
   RUNG wire#w2
      Move(in := #出库数量, out1 => #取出数量暂存)
   END_RUNG
   RUNG wire#w2
      Coil( #启动出库暂存."1" )
   END_RUNG
   RUNG wire#w1
      P_Contact(operand := #货物离开, bit := #货物离开_沿缓冲位."1")
      wire#w3
      Sub(in1 := #仓库货物数量, in2 := 1, out => #仓库货物数量)
   END_RUNG
   RUNG wire#w3
      Sub(in1 := #取出数量暂存, in2 := 1, out => #取出数量暂存)
   END_RUNG
   RUNG wire#w3
      { S7_Templates := "SrcType := Int" } GE_Contact(in1 := #取出数量暂存, in2 := 1)
      Coil( #启动出库暂存."2" )
   END_RUNG
   RUNG wire#w1
      Move(in := #仓库货物数量, out1 => #仓库位号输出)
   END_RUNG
   RUNG wire#powerrail
      Contact( #启动出库暂存."1" )
      wire#w4
      Coil( #启动出库 )
   END_RUNG
   RUNG wire#powerrail
      Contact( #启动出库暂存."2" )
   END_RUNG wire#w4
   RUNG wire#powerrail
      Contact( #出库完成 )
      R_Coil( #运行标志位.出库运行中 )
   END_RUNG
   RUNG wire#powerrail
      Contact( #出库模式 )
      { S7_Templates := "SrcType := Int" } EQ_Contact(in1 := #取出数量暂存, in2 := 0)
      wire#w5
      Coil( #完成出库或未启动出库 )
   END_RUNG
   RUNG wire#powerrail
      I_Contact( #出库模式 )
   END_RUNG wire#w5
   // the same network as SCL:
   #_w1 := #出库模式 AND #确认数量 AND (#出库数量 >= 1);
   IF #_w1 THEN
       #运行标志位.出库运行中 := TRUE;
       #取出数量暂存 := #出库数量;
   END_IF;
   #启动出库暂存."1" := #_w1;
   #_w2 := #出库模式 AND #货物离开 AND NOT #货物离开_沿缓冲位."1";   // rising edge of #货物离开
   #货物离开_沿缓冲位."1" := #货物离开;
   IF #_w2 THEN
       #仓库货物数量 := #仓库货物数量 - 1;
       #取出数量暂存 := #取出数量暂存 - 1;
   END_IF;
   #启动出库暂存."2" := #_w2 AND (#取出数量暂存 >= 1);
   IF #出库模式 THEN #仓库位号输出 := #仓库货物数量; END_IF;
   #启动出库 := #启动出库暂存."1" OR #启动出库暂存."2";
   IF #出库完成 THEN #运行标志位.出库运行中 := FALSE; END_IF;
   #完成出库或未启动出库 := (#出库模式 AND (#取出数量暂存 = 0)) OR NOT #出库模式;
END_REGION

REGION Network 3
   RUNG wire#powerrail
      { S7_Templates := "SrcType := Int" } EQ_Contact(in1 := #仓库货物数量, in2 := 54)
      Coil( #满仓 )
   END_RUNG
   RUNG wire#powerrail
      { S7_Templates := "SrcType := Int" } EQ_Contact(in1 := #仓库货物数量, in2 := 0)
      Coil( #无货 )
   END_RUNG
   // the same network as SCL:
   #满仓 := #仓库货物数量 = 54;
   #无货 := #仓库货物数量 = 0;
END_REGION
END_FUNCTION_BLOCK

FUNCTION_BLOCK "加工中心/传送带控制"   // FB4, LAD
{ S7_Optimized_Access := 'TRUE' }
VERSION : 0.1
   VAR_INPUT
      启动 : Bool;
      停止 : Bool;
      入料传感器 : Bool;
      出料传感器 : Bool;
      货箱到达传感器 : Bool;
   END_VAR
   VAR_OUTPUT
      加工中心启动 : Bool;
      加工中心停止 : Bool;
      加工中心生产上盖使能 : Bool;
      入料传送带 : Bool;
      出料传送带 : Bool;
      加工中 : Bool;
      货箱传送带 : Bool;
   END_VAR
   VAR
      加工中心运行步骤 : Int;
      加工中心沿缓冲位 : Struct
         "1" : Bool;
         "2" : Bool;
         "3" : Bool;
         "4" : Bool;
         "5" : Bool;
         "6" : Bool;
      END_STRUCT;
      货箱传送带沿缓冲位 : Struct
         "1" : Bool;
      END_STRUCT;
      运行标志位 : Bool;
      停止锁存位 : Bool;
   END_VAR
   VAR_TEMP   // added for the SCL form of the ladder/FBD networks
      _w1 : Bool;
      _w2 : Bool;
      _w3 : Bool;
      _w4 : Bool;
      _w5 : Bool;
      _w6 : Bool;
   END_VAR
BEGIN

REGION Network 1: 运料传送带
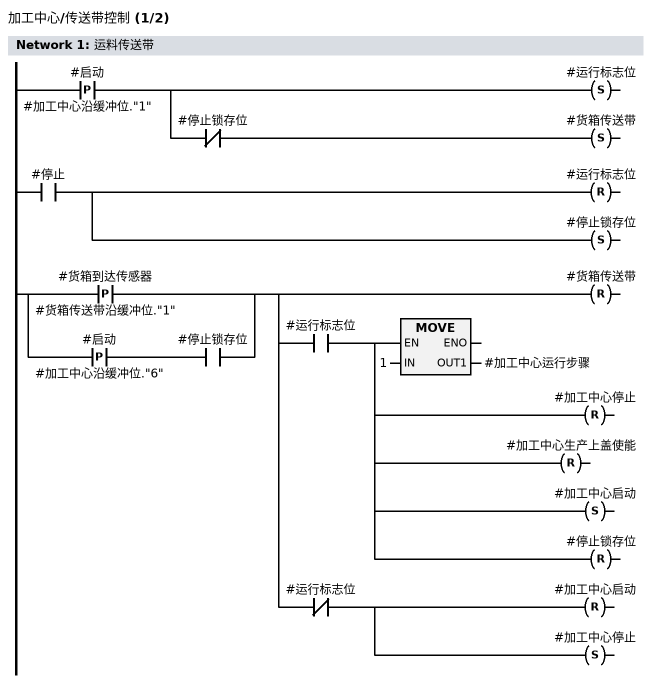
   RUNG wire#powerrail
      P_Contact(operand := #启动, bit := #加工中心沿缓冲位."1")
      wire#w1
      S_Coil( #运行标志位 )
   END_RUNG
   RUNG wire#w1
      I_Contact( #停止锁存位 )
      S_Coil( #货箱传送带 )
   END_RUNG
   RUNG wire#powerrail
      Contact( #停止 )
      wire#w2
      R_Coil( #运行标志位 )
   END_RUNG
   RUNG wire#w2
      S_Coil( #停止锁存位 )
   END_RUNG
   RUNG wire#powerrail
      P_Contact(operand := #货箱到达传感器, bit := #货箱传送带沿缓冲位."1")
      wire#w3
      R_Coil( #货箱传送带 )
   END_RUNG
   RUNG wire#powerrail
      P_Contact(operand := #启动, bit := #加工中心沿缓冲位."6")
      Contact( #停止锁存位 )
   END_RUNG wire#w3
   RUNG wire#w3
      Contact( #运行标志位 )
      wire#w4
      Move(in := 1, out1 => #加工中心运行步骤)
   END_RUNG
   RUNG wire#w4
      R_Coil( #加工中心停止 )
   END_RUNG
   RUNG wire#w4
      R_Coil( #加工中心生产上盖使能 )
   END_RUNG
   RUNG wire#w4
      S_Coil( #加工中心启动 )
   END_RUNG
   RUNG wire#w4
      R_Coil( #停止锁存位 )
   END_RUNG
   RUNG wire#w3
      I_Contact( #运行标志位 )
      wire#w5
      R_Coil( #加工中心启动 )
   END_RUNG
   RUNG wire#w5
      S_Coil( #加工中心停止 )
   END_RUNG
   // the same network as SCL:
   #_w1 := #启动 AND NOT #加工中心沿缓冲位."1";   // rising edge of #启动
   #加工中心沿缓冲位."1" := #启动;
   IF #_w1 THEN #运行标志位 := TRUE; END_IF;
   IF #_w1 AND NOT #停止锁存位 THEN #货箱传送带 := TRUE; END_IF;
   IF #停止 THEN
       #运行标志位 := FALSE;
       #停止锁存位 := TRUE;
   END_IF;
   #_w2 := #货箱到达传感器 AND NOT #货箱传送带沿缓冲位."1";   // rising edge of #货箱到达传感器
   #货箱传送带沿缓冲位."1" := #货箱到达传感器;
   #_w3 := #启动 AND NOT #加工中心沿缓冲位."6";   // rising edge of #启动
   #加工中心沿缓冲位."6" := #启动;
   #_w4 := #_w2 OR (#_w3 AND #停止锁存位);
   IF #_w4 THEN #货箱传送带 := FALSE; END_IF;
   IF #_w4 AND #运行标志位 THEN
       #加工中心运行步骤 := 1;
       #加工中心停止 := FALSE;
       #加工中心生产上盖使能 := FALSE;
       #加工中心启动 := TRUE;
       #停止锁存位 := FALSE;
   END_IF;
   IF #_w4 AND NOT #运行标志位 THEN
       #加工中心启动 := FALSE;
       #加工中心停止 := TRUE;
   END_IF;
END_REGION

REGION Network 2: 加工中心加工零件
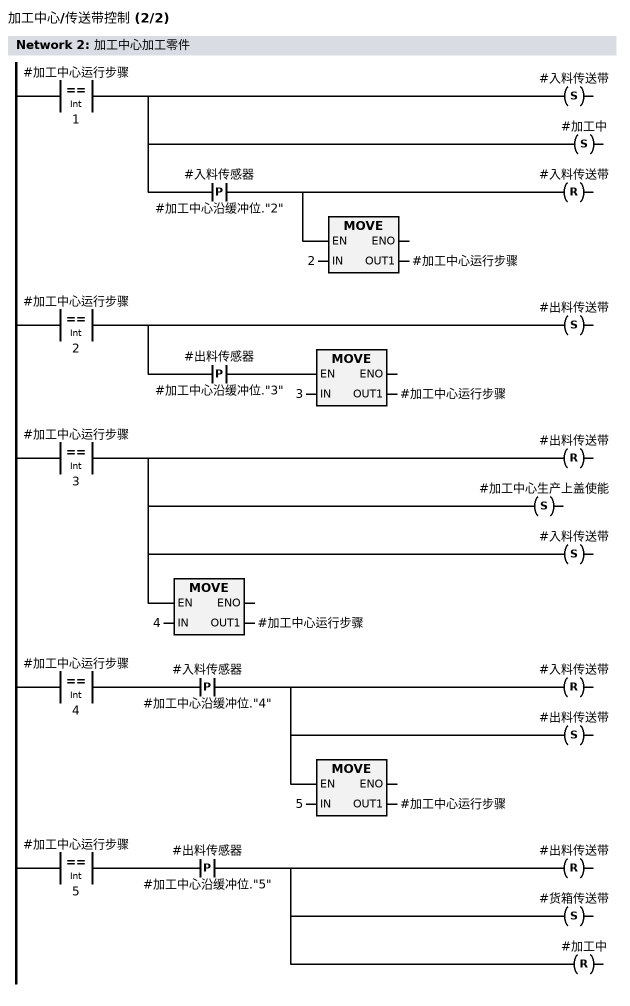
   RUNG wire#powerrail
      { S7_Templates := "SrcType := Int" } EQ_Contact(in1 := #加工中心运行步骤, in2 := 1)
      wire#w1
      S_Coil( #入料传送带 )
   END_RUNG
   RUNG wire#w1
      S_Coil( #加工中 )
   END_RUNG
   RUNG wire#w1
      P_Contact(operand := #入料传感器, bit := #加工中心沿缓冲位."2")
      wire#w2
      R_Coil( #入料传送带 )
   END_RUNG
   RUNG wire#w2
      Move(in := 2, out1 => #加工中心运行步骤)
   END_RUNG
   RUNG wire#powerrail
      { S7_Templates := "SrcType := Int" } EQ_Contact(in1 := #加工中心运行步骤, in2 := 2)
      wire#w3
      S_Coil( #出料传送带 )
   END_RUNG
   RUNG wire#w3
      P_Contact(operand := #出料传感器, bit := #加工中心沿缓冲位."3")
      Move(in := 3, out1 => #加工中心运行步骤)
   END_RUNG
   RUNG wire#powerrail
      { S7_Templates := "SrcType := Int" } EQ_Contact(in1 := #加工中心运行步骤, in2 := 3)
      wire#w4
      R_Coil( #出料传送带 )
   END_RUNG
   RUNG wire#w4
      S_Coil( #加工中心生产上盖使能 )
   END_RUNG
   RUNG wire#w4
      S_Coil( #入料传送带 )
   END_RUNG
   RUNG wire#w4
      Move(in := 4, out1 => #加工中心运行步骤)
   END_RUNG
   RUNG wire#powerrail
      { S7_Templates := "SrcType := Int" } EQ_Contact(in1 := #加工中心运行步骤, in2 := 4)
      P_Contact(operand := #入料传感器, bit := #加工中心沿缓冲位."4")
      wire#w5
      R_Coil( #入料传送带 )
   END_RUNG
   RUNG wire#w5
      S_Coil( #出料传送带 )
   END_RUNG
   RUNG wire#w5
      Move(in := 5, out1 => #加工中心运行步骤)
   END_RUNG
   RUNG wire#powerrail
      { S7_Templates := "SrcType := Int" } EQ_Contact(in1 := #加工中心运行步骤, in2 := 5)
      P_Contact(operand := #出料传感器, bit := #加工中心沿缓冲位."5")
      wire#w6
      R_Coil( #出料传送带 )
   END_RUNG
   RUNG wire#w6
      S_Coil( #货箱传送带 )
   END_RUNG
   RUNG wire#w6
      R_Coil( #加工中 )
   END_RUNG
   // the same network as SCL:
   #_w1 := #加工中心运行步骤 = 1;
   IF #_w1 THEN
       #入料传送带 := TRUE;
       #加工中 := TRUE;
   END_IF;
   #_w2 := #_w1 AND #入料传感器 AND NOT #加工中心沿缓冲位."2";   // rising edge of #入料传感器
   #加工中心沿缓冲位."2" := #入料传感器;
   IF #_w2 THEN
       #入料传送带 := FALSE;
       #加工中心运行步骤 := 2;
   END_IF;
   #_w3 := #加工中心运行步骤 = 2;
   IF #_w3 THEN #出料传送带 := TRUE; END_IF;
   #_w4 := #_w3 AND #出料传感器 AND NOT #加工中心沿缓冲位."3";   // rising edge of #出料传感器
   #加工中心沿缓冲位."3" := #出料传感器;
   IF #_w4 THEN #加工中心运行步骤 := 3; END_IF;
   IF #加工中心运行步骤 = 3 THEN
       #出料传送带 := FALSE;
       #加工中心生产上盖使能 := TRUE;
       #入料传送带 := TRUE;
       #加工中心运行步骤 := 4;
   END_IF;
   #_w5 := (#加工中心运行步骤 = 4) AND #入料传感器 AND NOT #加工中心沿缓冲位."4";   // rising edge of #入料传感器
   #加工中心沿缓冲位."4" := #入料传感器;
   IF #_w5 THEN
       #入料传送带 := FALSE;
       #出料传送带 := TRUE;
       #加工中心运行步骤 := 5;
   END_IF;
   #_w6 := (#加工中心运行步骤 = 5) AND #出料传感器 AND NOT #加工中心沿缓冲位."5";   // rising edge of #出料传感器
   #加工中心沿缓冲位."5" := #出料传感器;
   IF #_w6 THEN
       #出料传送带 := FALSE;
       #货箱传送带 := TRUE;
       #加工中 := FALSE;
   END_IF;
END_REGION
END_FUNCTION_BLOCK

FUNCTION_BLOCK "仓库/加工中心连接块"   // FB5, LAD
{ S7_Optimized_Access := 'TRUE' }
VERSION : 0.1
   VAR_INPUT
      仓库货物进入传感器 : Bool;
      入库完成 : Bool;
      入库模式 : Bool;
      货物到达传感器 : Bool;
      满仓信号 : Bool;
   END_VAR
   VAR_OUTPUT
      启动加工中心部分 : Bool;
      停止加工中心部分 : Bool;
      货物进入传送带 : Bool;
      末端传送带 : Bool;
   END_VAR
   VAR
      沿 : Struct
         "1" : Bool;
         "2" : Bool;
         "3" : Bool;
      END_STRUCT;
   END_VAR
   VAR_TEMP   // added for the SCL form of the ladder/FBD networks
      _w1 : Bool;
      _w2 : Bool;
      _w3 : Bool;
      _w4 : Bool;
   END_VAR
BEGIN

REGION Network 1
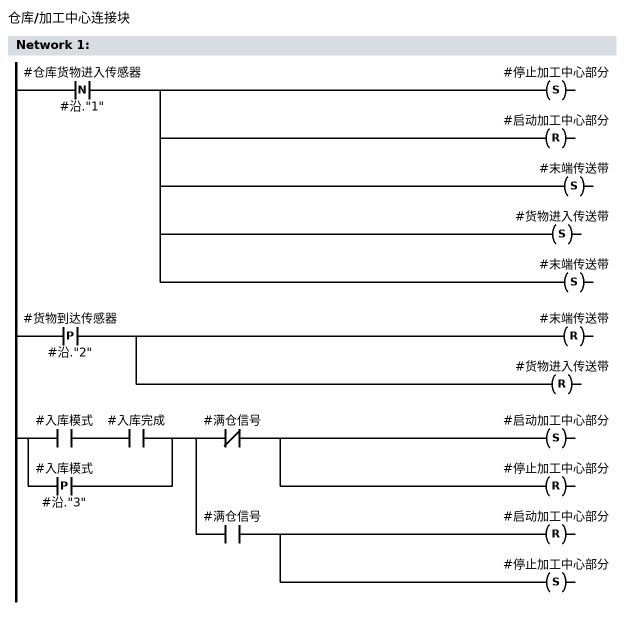
   RUNG wire#powerrail
      N_Contact(operand := #仓库货物进入传感器, bit := #沿."1")
      wire#w1
      S_Coil( #停止加工中心部分 )
   END_RUNG
   RUNG wire#w1
      R_Coil( #启动加工中心部分 )
   END_RUNG
   RUNG wire#w1
      S_Coil( #末端传送带 )
   END_RUNG
   RUNG wire#w1
      S_Coil( #货物进入传送带 )
   END_RUNG
   RUNG wire#w1
      S_Coil( #末端传送带 )
   END_RUNG
   RUNG wire#powerrail
      P_Contact(operand := #货物到达传感器, bit := #沿."2")
      wire#w2
      R_Coil( #末端传送带 )
   END_RUNG
   RUNG wire#w2
      R_Coil( #货物进入传送带 )
   END_RUNG
   RUNG wire#powerrail
      Contact( #入库模式 )
      Contact( #入库完成 )
      wire#w3
      I_Contact( #满仓信号 )
      wire#w4
      S_Coil( #启动加工中心部分 )
   END_RUNG
   RUNG wire#powerrail
      P_Contact(operand := #入库模式, bit := #沿."3")
   END_RUNG wire#w3
   RUNG wire#w4
      R_Coil( #停止加工中心部分 )
   END_RUNG
   RUNG wire#w3
      Contact( #满仓信号 )
      wire#w5
      R_Coil( #启动加工中心部分 )
   END_RUNG
   RUNG wire#w5
      S_Coil( #停止加工中心部分 )
   END_RUNG
   // the same network as SCL:
   #_w1 := NOT #仓库货物进入传感器 AND #沿."1";   // falling edge of #仓库货物进入传感器
   #沿."1" := #仓库货物进入传感器;
   IF #_w1 THEN
       #停止加工中心部分 := TRUE;
       #启动加工中心部分 := FALSE;
       #末端传送带 := TRUE;
       #货物进入传送带 := TRUE;
       #末端传送带 := TRUE;
   END_IF;
   #_w2 := #货物到达传感器 AND NOT #沿."2";   // rising edge of #货物到达传感器
   #沿."2" := #货物到达传感器;
   IF #_w2 THEN
       #末端传送带 := FALSE;
       #货物进入传送带 := FALSE;
   END_IF;
   #_w3 := #入库模式 AND NOT #沿."3";   // rising edge of #入库模式
   #沿."3" := #入库模式;
   #_w4 := (#入库模式 AND #入库完成) OR #_w3;
   IF #_w4 AND NOT #满仓信号 THEN
       #启动加工中心部分 := TRUE;
       #停止加工中心部分 := FALSE;
   END_IF;
   IF #_w4 AND #满仓信号 THEN
       #启动加工中心部分 := FALSE;
       #停止加工中心部分 := TRUE;
   END_IF;
END_REGION
END_FUNCTION_BLOCK

FUNCTION_BLOCK "汇总块"   // FB6, LAD
{ S7_Optimized_Access := 'TRUE' }
VERSION : 0.1
   VAR_INPUT
      出库模式 : Bool;
      入库模式 : Bool;
      出库数量设置 : Int;
      确认出库数量 : Bool;
      码货龙门运行中 : Bool;
      取货器左移到达 : Bool;
      取货器右移到达 : Bool;
      取货器归位 : Bool;
      仓取货器运行中 : Bool;
      货物到达传感器 : Bool;
      货物进入传感器 : Bool;
      货物离开传感器 : Bool;
      加工中心入料传感器 : Bool;
      加工中心出料传感器 : Bool;
      货箱到达传感器 : Bool;
   END_VAR
   VAR_OUTPUT
      目标仓位 : DInt;
      取货器左移 : Bool;
      取货器右移 : Bool;
      取货器上升 : Bool;
      货物进入传送带 : Bool;
      传送带末端 : Bool;
      加工中心启动 : Bool;
      加工中心停止 : Bool;
      加工中心加工上盖使能 : Bool;
      加工中心入料传送带 : Bool;
      进货传送带 : Bool;
      加工中心出料传送带 : Bool;
      出库完成或未启用出库模式 : Bool;
      入库完成 : Bool;
      满仓信号 : Bool;
   END_VAR
   VAR_IN_OUT
      仓库数据 : Int;
   END_VAR
   VAR
      "加工中心/传送带控制_Instance" : "加工中心/传送带控制";
      进出库调度_Instance : "进出库调度";
      龙门码货机_Instance : "龙门码货机";
      "仓库/加工中心连接块_Instance" : "仓库/加工中心连接块";
   END_VAR
   VAR_TEMP   // added for the SCL form of the ladder/FBD networks
      _w1 : Bool;
   END_VAR
BEGIN

REGION Network 1
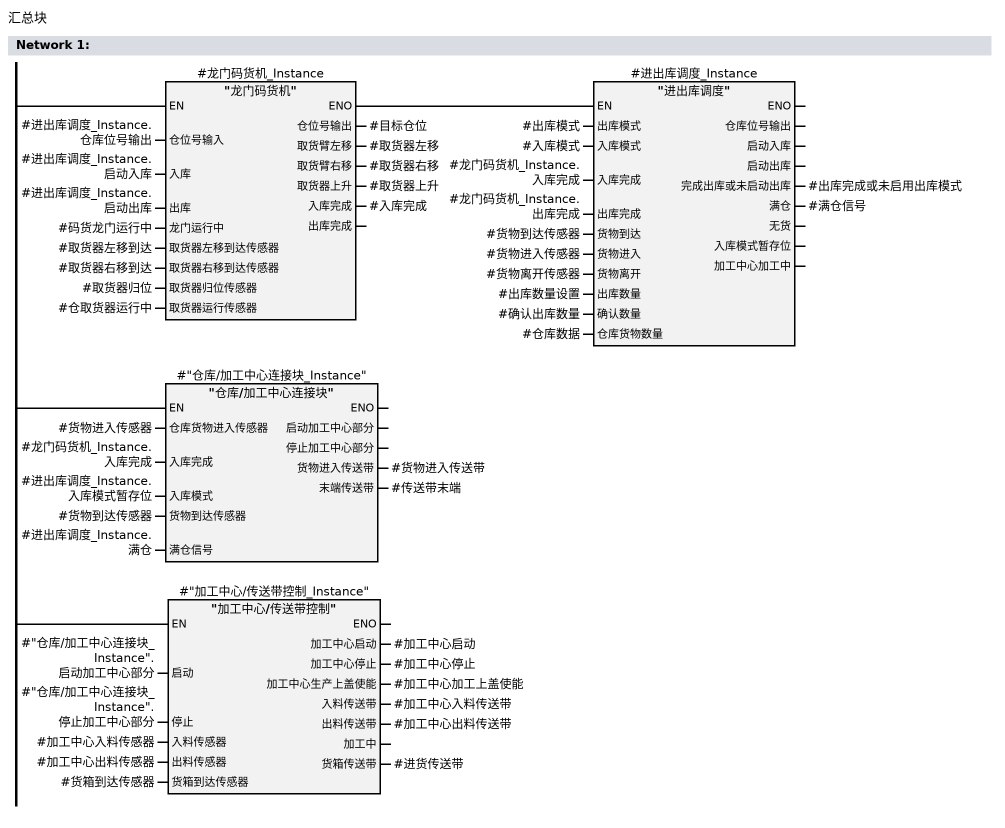
   RUNG wire#powerrail
      #龙门码货机_Instance(仓位号输入 := #进出库调度_Instance.仓库位号输出, 入库 := #进出库调度_Instance.启动入库, 出库 := #进出库调度_Instance.启动出库, 龙门运行中 := #码货龙门运行中, 取货器左移到达传感器 := #取货器左移到达, 取货器右移到达传感器 := #取货器右移到达, 取货器归位传感器 := #取货器归位, 取货器运行传感器 := #仓取货器运行中, 仓位号输出 => #目标仓位, 取货臂左移 => #取货器左移, 取货臂右移 => #取货器右移, 取货器上升 => #取货器上升, 入库完成 => #入库完成, 出库完成 =>)
      #进出库调度_Instance(出库模式 := #出库模式, 入库模式 := #入库模式, 入库完成 := #龙门码货机_Instance.入库完成, 出库完成 := #龙门码货机_Instance.出库完成, 货物到达 := #货物到达传感器, 货物进入 := #货物进入传感器, 货物离开 := #货物离开传感器, 出库数量 := #出库数量设置, 确认数量 := #确认出库数量, 仓库货物数量 := #仓库数据, 仓库位号输出 =>, 启动入库 =>, 启动出库 =>, 完成出库或未启动出库 => #出库完成或未启用出库模式, 满仓 => #满仓信号, 无货 =>, 入库模式暂存位 =>, 加工中心加工中 =>)
   END_RUNG
   RUNG wire#powerrail
      #"仓库/加工中心连接块_Instance"(仓库货物进入传感器 := #货物进入传感器, 入库完成 := #龙门码货机_Instance.入库完成, 入库模式 := #进出库调度_Instance.入库模式暂存位, 货物到达传感器 := #货物到达传感器, 满仓信号 := #进出库调度_Instance.满仓, 启动加工中心部分 =>, 停止加工中心部分 =>, 货物进入传送带 => #货物进入传送带, 末端传送带 => #传送带末端)
   END_RUNG
   RUNG wire#powerrail
      #"加工中心/传送带控制_Instance"(启动 := #"仓库/加工中心连接块_Instance".启动加工中心部分, 停止 := #"仓库/加工中心连接块_Instance".停止加工中心部分, 入料传感器 := #加工中心入料传感器, 出料传感器 := #加工中心出料传感器, 货箱到达传感器 := #货箱到达传感器, 加工中心启动 => #加工中心启动, 加工中心停止 => #加工中心停止, 加工中心生产上盖使能 => #加工中心加工上盖使能, 入料传送带 => #加工中心入料传送带, 出料传送带 => #加工中心出料传送带, 加工中 =>, 货箱传送带 => #进货传送带)
   END_RUNG
   // the same network as SCL:
   #龙门码货机_Instance(仓位号输入 := #进出库调度_Instance.仓库位号输出,   // "龙门码货机"
                   入库 := #进出库调度_Instance.启动入库,
                   出库 := #进出库调度_Instance.启动出库,
                   龙门运行中 := #码货龙门运行中,
                   取货器左移到达传感器 := #取货器左移到达,
                   取货器右移到达传感器 := #取货器右移到达,
                   取货器归位传感器 := #取货器归位,
                   取货器运行传感器 := #仓取货器运行中,
                   仓位号输出 => #目标仓位,
                   取货臂左移 => #取货器左移,
                   取货臂右移 => #取货器右移,
                   取货器上升 => #取货器上升,
                   入库完成 => #入库完成,
                   ENO => #_w1);
   IF #_w1 THEN
       #进出库调度_Instance(出库模式 := #出库模式,   // "进出库调度"
                       入库模式 := #入库模式,
                       入库完成 := #龙门码货机_Instance.入库完成,
                       出库完成 := #龙门码货机_Instance.出库完成,
                       货物到达 := #货物到达传感器,
                       货物进入 := #货物进入传感器,
                       货物离开 := #货物离开传感器,
                       出库数量 := #出库数量设置,
                       确认数量 := #确认出库数量,
                       仓库货物数量 := #仓库数据,
                       完成出库或未启动出库 => #出库完成或未启用出库模式,
                       满仓 => #满仓信号);
   END_IF;
   #"仓库/加工中心连接块_Instance"(仓库货物进入传感器 := #货物进入传感器,   // "仓库/加工中心连接块"
                          入库完成 := #龙门码货机_Instance.入库完成,
                          入库模式 := #进出库调度_Instance.入库模式暂存位,
                          货物到达传感器 := #货物到达传感器,
                          满仓信号 := #进出库调度_Instance.满仓,
                          货物进入传送带 => #货物进入传送带,
                          末端传送带 => #传送带末端);
   #"加工中心/传送带控制_Instance"(启动 := #"仓库/加工中心连接块_Instance".启动加工中心部分,   // "加工中心/传送带控制"
                          停止 := #"仓库/加工中心连接块_Instance".停止加工中心部分,
                          入料传感器 := #加工中心入料传感器,
                          出料传感器 := #加工中心出料传感器,
                          货箱到达传感器 := #货箱到达传感器,
                          加工中心启动 => #加工中心启动,
                          加工中心停止 => #加工中心停止,
                          加工中心生产上盖使能 => #加工中心加工上盖使能,
                          入料传送带 => #加工中心入料传送带,
                          出料传送带 => #加工中心出料传送带,
                          货箱传送带 => #进货传送带);
END_REGION
END_FUNCTION_BLOCK

FUNCTION "自动运行" : Void   // FC1, LAD
{ S7_Optimized_Access := 'TRUE' }
VERSION : 0.1
   VAR_TEMP   // added for the SCL form of the ladder/FBD networks
      _w1 : Bool;
      _w2 : Bool;
      _w3 : Bool;
      _w4 : Bool;
      _w5 : Bool;
      _w6 : Bool;
      _w7 : Bool;
      _w8 : Bool;
      _w9 : Bool;
      _w10 : Bool;
   END_VAR
BEGIN

REGION Network 2: 仓库控制
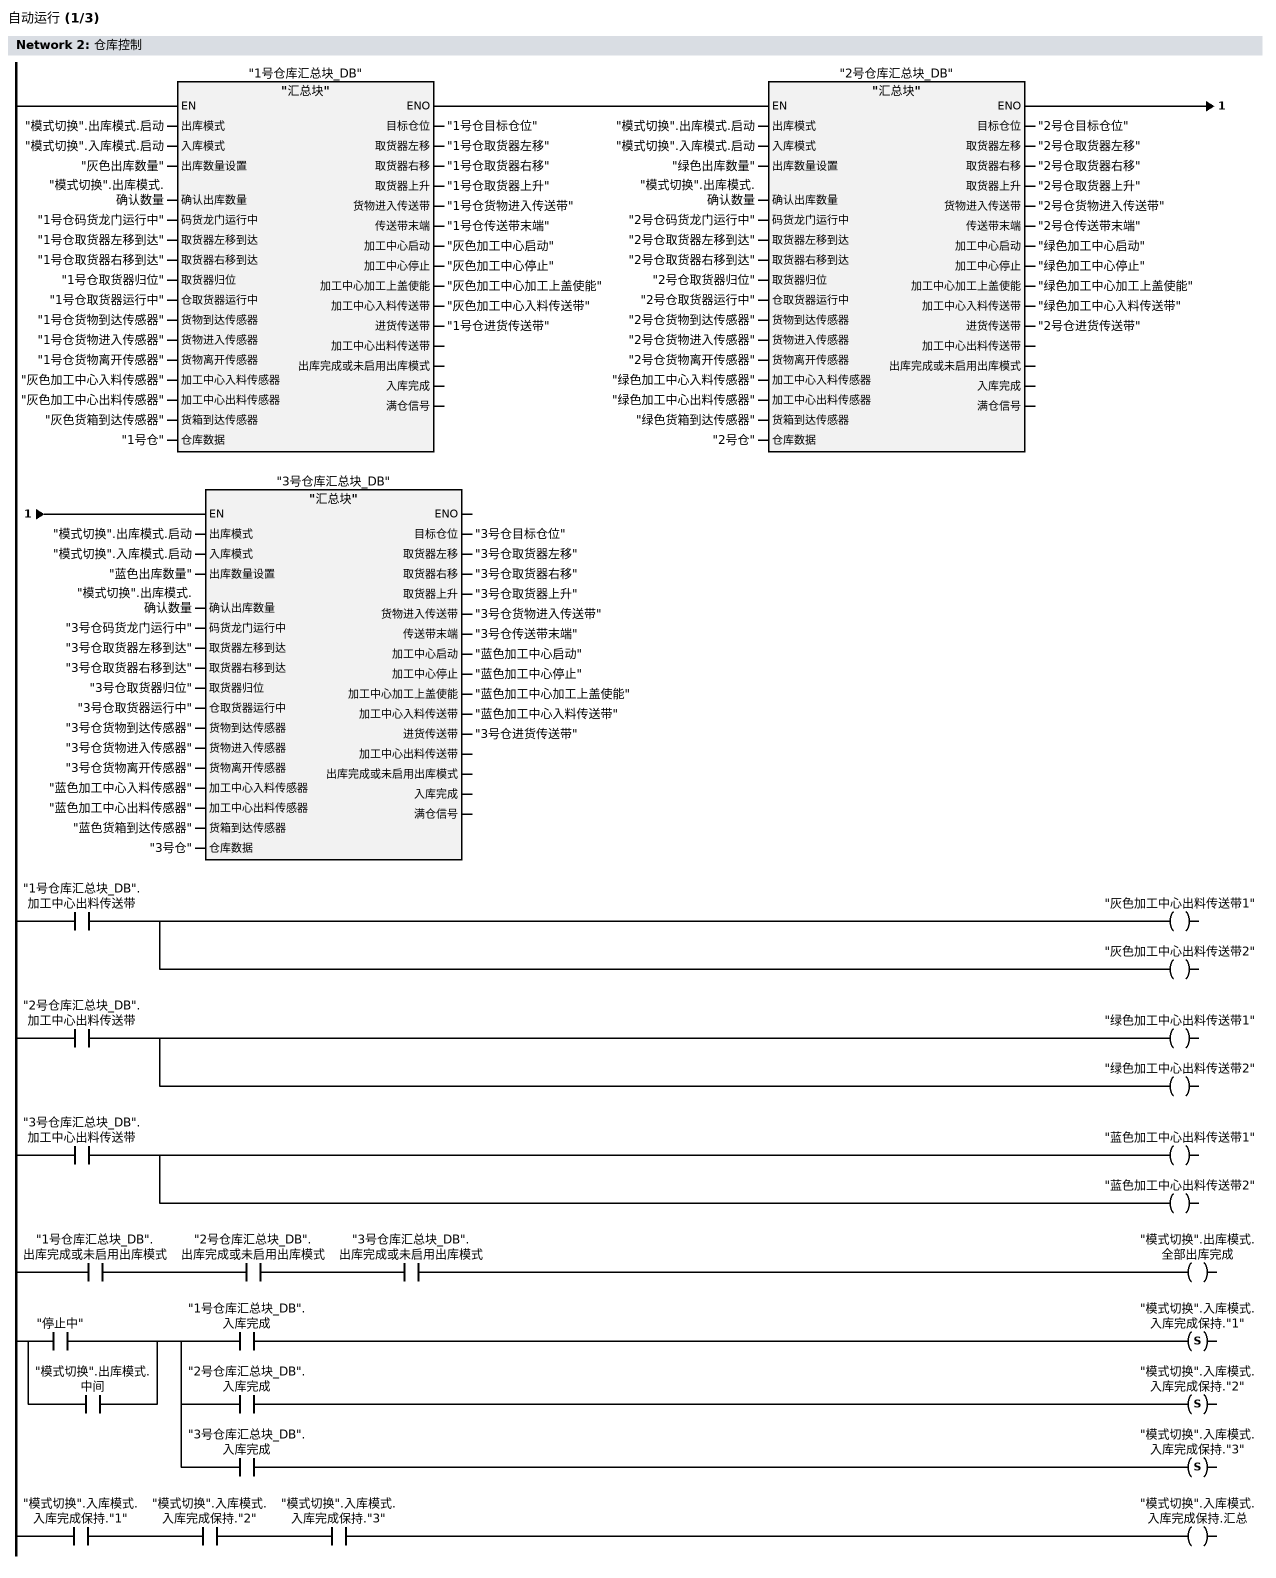
   RUNG wire#powerrail
      "1号仓库汇总块_DB"(出库模式 := "模式切换".出库模式.启动, 入库模式 := "模式切换".入库模式.启动, 出库数量设置 := "灰色出库数量", 确认出库数量 := "模式切换".出库模式.确认数量, 码货龙门运行中 := "1号仓码货龙门运行中", 取货器左移到达 := "1号仓取货器左移到达", 取货器右移到达 := "1号仓取货器右移到达", 取货器归位 := "1号仓取货器归位", 仓取货器运行中 := "1号仓取货器运行中", 货物到达传感器 := "1号仓货物到达传感器", 货物进入传感器 := "1号仓货物进入传感器", 货物离开传感器 := "1号仓货物离开传感器", 加工中心入料传感器 := "灰色加工中心入料传感器", 加工中心出料传感器 := "灰色加工中心出料传感器", 货箱到达传感器 := "灰色货箱到达传感器", 仓库数据 := "1号仓", 目标仓位 => "1号仓目标仓位", 取货器左移 => "1号仓取货器左移", 取货器右移 => "1号仓取货器右移", 取货器上升 => "1号仓取货器上升", 货物进入传送带 => "1号仓货物进入传送带", 传送带末端 => "1号仓传送带末端", 加工中心启动 => "灰色加工中心启动", 加工中心停止 => "灰色加工中心停止", 加工中心加工上盖使能 => "灰色加工中心加工上盖使能", 加工中心入料传送带 => "灰色加工中心入料传送带", 进货传送带 => "1号仓进货传送带", 加工中心出料传送带 =>, 出库完成或未启用出库模式 =>, 入库完成 =>, 满仓信号 =>)
      "2号仓库汇总块_DB"(出库模式 := "模式切换".出库模式.启动, 入库模式 := "模式切换".入库模式.启动, 出库数量设置 := "绿色出库数量", 确认出库数量 := "模式切换".出库模式.确认数量, 码货龙门运行中 := "2号仓码货龙门运行中", 取货器左移到达 := "2号仓取货器左移到达", 取货器右移到达 := "2号仓取货器右移到达", 取货器归位 := "2号仓取货器归位", 仓取货器运行中 := "2号仓取货器运行中", 货物到达传感器 := "2号仓货物到达传感器", 货物进入传感器 := "2号仓货物进入传感器", 货物离开传感器 := "2号仓货物离开传感器", 加工中心入料传感器 := "绿色加工中心入料传感器", 加工中心出料传感器 := "绿色加工中心出料传感器", 货箱到达传感器 := "绿色货箱到达传感器", 仓库数据 := "2号仓", 目标仓位 => "2号仓目标仓位", 取货器左移 => "2号仓取货器左移", 取货器右移 => "2号仓取货器右移", 取货器上升 => "2号仓取货器上升", 货物进入传送带 => "2号仓货物进入传送带", 传送带末端 => "2号仓传送带末端", 加工中心启动 => "绿色加工中心启动", 加工中心停止 => "绿色加工中心停止", 加工中心加工上盖使能 => "绿色加工中心加工上盖使能", 加工中心入料传送带 => "绿色加工中心入料传送带", 进货传送带 => "2号仓进货传送带", 加工中心出料传送带 =>, 出库完成或未启用出库模式 =>, 入库完成 =>, 满仓信号 =>)
      "3号仓库汇总块_DB"(出库模式 := "模式切换".出库模式.启动, 入库模式 := "模式切换".入库模式.启动, 出库数量设置 := "蓝色出库数量", 确认出库数量 := "模式切换".出库模式.确认数量, 码货龙门运行中 := "3号仓码货龙门运行中", 取货器左移到达 := "3号仓取货器左移到达", 取货器右移到达 := "3号仓取货器右移到达", 取货器归位 := "3号仓取货器归位", 仓取货器运行中 := "3号仓取货器运行中", 货物到达传感器 := "3号仓货物到达传感器", 货物进入传感器 := "3号仓货物进入传感器", 货物离开传感器 := "3号仓货物离开传感器", 加工中心入料传感器 := "蓝色加工中心入料传感器", 加工中心出料传感器 := "蓝色加工中心出料传感器", 货箱到达传感器 := "蓝色货箱到达传感器", 仓库数据 := "3号仓", 目标仓位 => "3号仓目标仓位", 取货器左移 => "3号仓取货器左移", 取货器右移 => "3号仓取货器右移", 取货器上升 => "3号仓取货器上升", 货物进入传送带 => "3号仓货物进入传送带", 传送带末端 => "3号仓传送带末端", 加工中心启动 => "蓝色加工中心启动", 加工中心停止 => "蓝色加工中心停止", 加工中心加工上盖使能 => "蓝色加工中心加工上盖使能", 加工中心入料传送带 => "蓝色加工中心入料传送带", 进货传送带 => "3号仓进货传送带", 加工中心出料传送带 =>, 出库完成或未启用出库模式 =>, 入库完成 =>, 满仓信号 =>)
   END_RUNG
   RUNG wire#powerrail
      Contact( "1号仓库汇总块_DB".加工中心出料传送带 )
      wire#w1
      Coil( "灰色加工中心出料传送带1" )
   END_RUNG
   RUNG wire#w1
      Coil( "灰色加工中心出料传送带2" )
   END_RUNG
   RUNG wire#powerrail
      Contact( "2号仓库汇总块_DB".加工中心出料传送带 )
      wire#w2
      Coil( "绿色加工中心出料传送带1" )
   END_RUNG
   RUNG wire#w2
      Coil( "绿色加工中心出料传送带2" )
   END_RUNG
   RUNG wire#powerrail
      Contact( "3号仓库汇总块_DB".加工中心出料传送带 )
      wire#w3
      Coil( "蓝色加工中心出料传送带1" )
   END_RUNG
   RUNG wire#w3
      Coil( "蓝色加工中心出料传送带2" )
   END_RUNG
   RUNG wire#powerrail
      Contact( "1号仓库汇总块_DB".出库完成或未启用出库模式 )
      Contact( "2号仓库汇总块_DB".出库完成或未启用出库模式 )
      Contact( "3号仓库汇总块_DB".出库完成或未启用出库模式 )
      Coil( "模式切换".出库模式.全部出库完成 )
   END_RUNG
   RUNG wire#powerrail
      Contact( "停止中" )
      wire#w4
      Contact( "1号仓库汇总块_DB".入库完成 )
      S_Coil( "模式切换".入库模式.入库完成保持."1" )
   END_RUNG
   RUNG wire#powerrail
      Contact( "模式切换".出库模式.中间 )
   END_RUNG wire#w4
   RUNG wire#w4
      Contact( "2号仓库汇总块_DB".入库完成 )
      S_Coil( "模式切换".入库模式.入库完成保持."2" )
   END_RUNG
   RUNG wire#w4
      Contact( "3号仓库汇总块_DB".入库完成 )
      S_Coil( "模式切换".入库模式.入库完成保持."3" )
   END_RUNG
   RUNG wire#powerrail
      Contact( "模式切换".入库模式.入库完成保持."1" )
      Contact( "模式切换".入库模式.入库完成保持."2" )
      Contact( "模式切换".入库模式.入库完成保持."3" )
      Coil( "模式切换".入库模式.入库完成保持.汇总 )
   END_RUNG
   // the same network as SCL:
   "1号仓库汇总块_DB"(出库模式 := "模式切换".出库模式.启动,   // "汇总块"
                入库模式 := "模式切换".入库模式.启动,
                出库数量设置 := "灰色出库数量",
                确认出库数量 := "模式切换".出库模式.确认数量,
                码货龙门运行中 := "1号仓码货龙门运行中",
                取货器左移到达 := "1号仓取货器左移到达",
                取货器右移到达 := "1号仓取货器右移到达",
                取货器归位 := "1号仓取货器归位",
                仓取货器运行中 := "1号仓取货器运行中",
                货物到达传感器 := "1号仓货物到达传感器",
                货物进入传感器 := "1号仓货物进入传感器",
                货物离开传感器 := "1号仓货物离开传感器",
                加工中心入料传感器 := "灰色加工中心入料传感器",
                加工中心出料传感器 := "灰色加工中心出料传感器",
                货箱到达传感器 := "灰色货箱到达传感器",
                仓库数据 := "1号仓",
                目标仓位 => "1号仓目标仓位",
                取货器左移 => "1号仓取货器左移",
                取货器右移 => "1号仓取货器右移",
                取货器上升 => "1号仓取货器上升",
                货物进入传送带 => "1号仓货物进入传送带",
                传送带末端 => "1号仓传送带末端",
                加工中心启动 => "灰色加工中心启动",
                加工中心停止 => "灰色加工中心停止",
                加工中心加工上盖使能 => "灰色加工中心加工上盖使能",
                加工中心入料传送带 => "灰色加工中心入料传送带",
                进货传送带 => "1号仓进货传送带",
                ENO => #_w1);
   "2号仓库汇总块_DB"(EN := #_w1,   // "汇总块"
                出库模式 := "模式切换".出库模式.启动,
                入库模式 := "模式切换".入库模式.启动,
                出库数量设置 := "绿色出库数量",
                确认出库数量 := "模式切换".出库模式.确认数量,
                码货龙门运行中 := "2号仓码货龙门运行中",
                取货器左移到达 := "2号仓取货器左移到达",
                取货器右移到达 := "2号仓取货器右移到达",
                取货器归位 := "2号仓取货器归位",
                仓取货器运行中 := "2号仓取货器运行中",
                货物到达传感器 := "2号仓货物到达传感器",
                货物进入传感器 := "2号仓货物进入传感器",
                货物离开传感器 := "2号仓货物离开传感器",
                加工中心入料传感器 := "绿色加工中心入料传感器",
                加工中心出料传感器 := "绿色加工中心出料传感器",
                货箱到达传感器 := "绿色货箱到达传感器",
                仓库数据 := "2号仓",
                目标仓位 => "2号仓目标仓位",
                取货器左移 => "2号仓取货器左移",
                取货器右移 => "2号仓取货器右移",
                取货器上升 => "2号仓取货器上升",
                货物进入传送带 => "2号仓货物进入传送带",
                传送带末端 => "2号仓传送带末端",
                加工中心启动 => "绿色加工中心启动",
                加工中心停止 => "绿色加工中心停止",
                加工中心加工上盖使能 => "绿色加工中心加工上盖使能",
                加工中心入料传送带 => "绿色加工中心入料传送带",
                进货传送带 => "2号仓进货传送带",
                ENO => #_w2);
   IF #_w2 THEN
       "3号仓库汇总块_DB"(出库模式 := "模式切换".出库模式.启动,   // "汇总块"
                    入库模式 := "模式切换".入库模式.启动,
                    出库数量设置 := "蓝色出库数量",
                    确认出库数量 := "模式切换".出库模式.确认数量,
                    码货龙门运行中 := "3号仓码货龙门运行中",
                    取货器左移到达 := "3号仓取货器左移到达",
                    取货器右移到达 := "3号仓取货器右移到达",
                    取货器归位 := "3号仓取货器归位",
                    仓取货器运行中 := "3号仓取货器运行中",
                    货物到达传感器 := "3号仓货物到达传感器",
                    货物进入传感器 := "3号仓货物进入传感器",
                    货物离开传感器 := "3号仓货物离开传感器",
                    加工中心入料传感器 := "蓝色加工中心入料传感器",
                    加工中心出料传感器 := "蓝色加工中心出料传感器",
                    货箱到达传感器 := "蓝色货箱到达传感器",
                    仓库数据 := "3号仓",
                    目标仓位 => "3号仓目标仓位",
                    取货器左移 => "3号仓取货器左移",
                    取货器右移 => "3号仓取货器右移",
                    取货器上升 => "3号仓取货器上升",
                    货物进入传送带 => "3号仓货物进入传送带",
                    传送带末端 => "3号仓传送带末端",
                    加工中心启动 => "蓝色加工中心启动",
                    加工中心停止 => "蓝色加工中心停止",
                    加工中心加工上盖使能 => "蓝色加工中心加工上盖使能",
                    加工中心入料传送带 => "蓝色加工中心入料传送带",
                    进货传送带 => "3号仓进货传送带");
   END_IF;
   "灰色加工中心出料传送带1" := "1号仓库汇总块_DB".加工中心出料传送带;
   "灰色加工中心出料传送带2" := "1号仓库汇总块_DB".加工中心出料传送带;
   "绿色加工中心出料传送带1" := "2号仓库汇总块_DB".加工中心出料传送带;
   "绿色加工中心出料传送带2" := "2号仓库汇总块_DB".加工中心出料传送带;
   "蓝色加工中心出料传送带1" := "3号仓库汇总块_DB".加工中心出料传送带;
   "蓝色加工中心出料传送带2" := "3号仓库汇总块_DB".加工中心出料传送带;
   "模式切换".出库模式.全部出库完成 := "1号仓库汇总块_DB".出库完成或未启用出库模式 AND "2号仓库汇总块_DB".出库完成或未启用出库模式 AND "3号仓库汇总块_DB".出库完成或未启用出库模式;
   #_w3 := "停止中" OR "模式切换".出库模式.中间;
   IF #_w3 AND "1号仓库汇总块_DB".入库完成 THEN "模式切换".入库模式.入库完成保持."1" := TRUE; END_IF;
   IF #_w3 AND "2号仓库汇总块_DB".入库完成 THEN "模式切换".入库模式.入库完成保持."2" := TRUE; END_IF;
   IF #_w3 AND "3号仓库汇总块_DB".入库完成 THEN "模式切换".入库模式.入库完成保持."3" := TRUE; END_IF;
   "模式切换".入库模式.入库完成保持.汇总 := "模式切换".入库模式.入库完成保持."1" AND "模式切换".入库模式.入库完成保持."2" AND "模式切换".入库模式.入库完成保持."3";
END_REGION

REGION Network 3: 模式切换
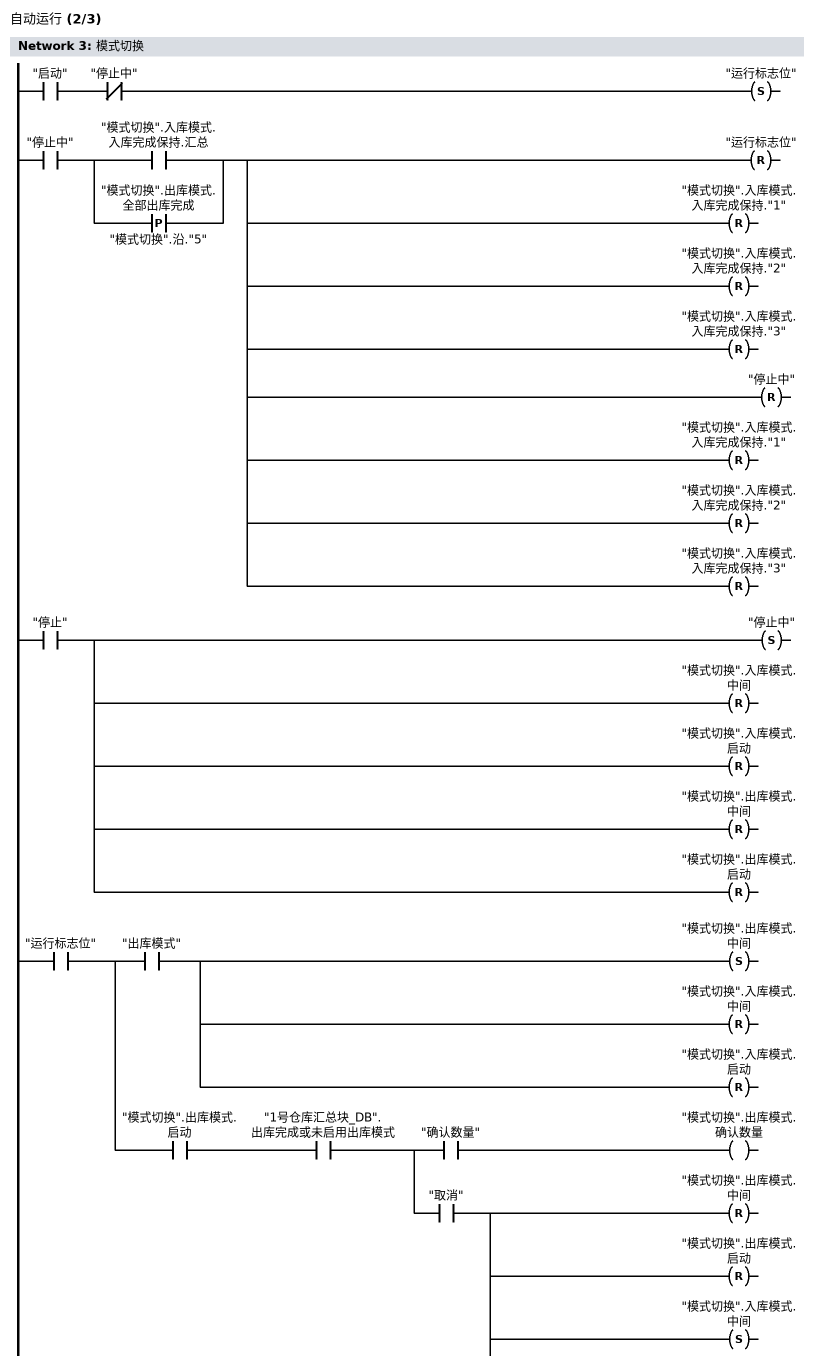
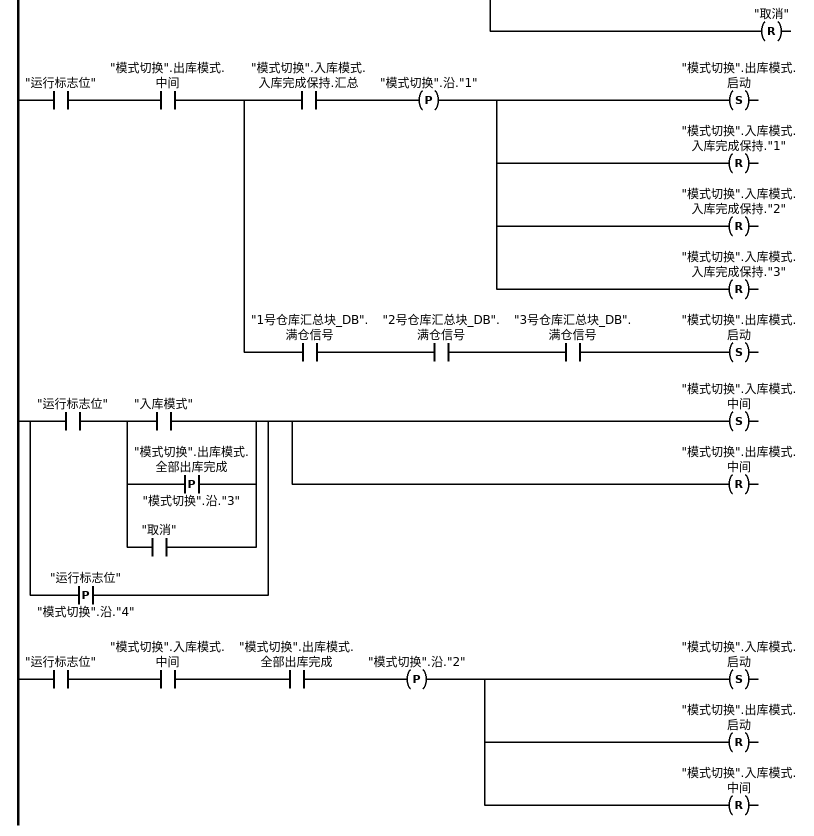
   RUNG wire#powerrail
      Contact( "启动" )
      I_Contact( "停止中" )
      S_Coil( "运行标志位" )
   END_RUNG
   RUNG wire#powerrail
      Contact( "停止中" )
      wire#w1
      Contact( "模式切换".入库模式.入库完成保持.汇总 )
      wire#w2
      R_Coil( "运行标志位" )
   END_RUNG
   RUNG wire#w1
      P_Contact(operand := "模式切换".出库模式.全部出库完成, bit := "模式切换".沿."5")
   END_RUNG wire#w2
   RUNG wire#w2
      R_Coil( "模式切换".入库模式.入库完成保持."1" )
   END_RUNG
   RUNG wire#w2
      R_Coil( "模式切换".入库模式.入库完成保持."2" )
   END_RUNG
   RUNG wire#w2
      R_Coil( "模式切换".入库模式.入库完成保持."3" )
   END_RUNG
   RUNG wire#w2
      R_Coil( "停止中" )
   END_RUNG
   RUNG wire#w2
      R_Coil( "模式切换".入库模式.入库完成保持."1" )
   END_RUNG
   RUNG wire#w2
      R_Coil( "模式切换".入库模式.入库完成保持."2" )
   END_RUNG
   RUNG wire#w2
      R_Coil( "模式切换".入库模式.入库完成保持."3" )
   END_RUNG
   RUNG wire#powerrail
      Contact( "停止" )
      wire#w3
      S_Coil( "停止中" )
   END_RUNG
   RUNG wire#w3
      R_Coil( "模式切换".入库模式.中间 )
   END_RUNG
   RUNG wire#w3
      R_Coil( "模式切换".入库模式.启动 )
   END_RUNG
   RUNG wire#w3
      R_Coil( "模式切换".出库模式.中间 )
   END_RUNG
   RUNG wire#w3
      R_Coil( "模式切换".出库模式.启动 )
   END_RUNG
   RUNG wire#powerrail
      Contact( "运行标志位" )
      wire#w4
      Contact( "出库模式" )
      wire#w5
      S_Coil( "模式切换".出库模式.中间 )
   END_RUNG
   RUNG wire#w5
      R_Coil( "模式切换".入库模式.中间 )
   END_RUNG
   RUNG wire#w5
      R_Coil( "模式切换".入库模式.启动 )
   END_RUNG
   RUNG wire#w4
      Contact( "模式切换".出库模式.启动 )
      Contact( "1号仓库汇总块_DB".出库完成或未启用出库模式 )
      wire#w6
      Contact( "确认数量" )
      Coil( "模式切换".出库模式.确认数量 )
   END_RUNG
   RUNG wire#w6
      Contact( "取消" )
      wire#w7
      R_Coil( "模式切换".出库模式.中间 )
   END_RUNG
   RUNG wire#w7
      R_Coil( "模式切换".出库模式.启动 )
   END_RUNG
   RUNG wire#w7
      S_Coil( "模式切换".入库模式.中间 )
   END_RUNG
   RUNG wire#w7
      R_Coil( "取消" )
   END_RUNG
   RUNG wire#powerrail
      Contact( "运行标志位" )
      Contact( "模式切换".出库模式.中间 )
      wire#w8
      Contact( "模式切换".入库模式.入库完成保持.汇总 )
      P_Trig( "模式切换".沿."1" )
      wire#w9
      S_Coil( "模式切换".出库模式.启动 )
   END_RUNG
   RUNG wire#w9
      R_Coil( "模式切换".入库模式.入库完成保持."1" )
   END_RUNG
   RUNG wire#w9
      R_Coil( "模式切换".入库模式.入库完成保持."2" )
   END_RUNG
   RUNG wire#w9
      R_Coil( "模式切换".入库模式.入库完成保持."3" )
   END_RUNG
   RUNG wire#w8
      Contact( "1号仓库汇总块_DB".满仓信号 )
      Contact( "2号仓库汇总块_DB".满仓信号 )
      Contact( "3号仓库汇总块_DB".满仓信号 )
      S_Coil( "模式切换".出库模式.启动 )
   END_RUNG
   RUNG wire#powerrail
      Contact( "运行标志位" )
      wire#w10
      Contact( "入库模式" )
      wire#w11
      S_Coil( "模式切换".入库模式.中间 )
   END_RUNG
   RUNG wire#w10
      P_Contact(operand := "模式切换".出库模式.全部出库完成, bit := "模式切换".沿."3")
   END_RUNG wire#w11
   RUNG wire#w10
      Contact( "取消" )
   END_RUNG wire#w11
   RUNG wire#powerrail
      P_Contact(operand := "运行标志位", bit := "模式切换".沿."4")
   END_RUNG wire#w11
   RUNG wire#w11
      R_Coil( "模式切换".出库模式.中间 )
   END_RUNG
   RUNG wire#powerrail
      Contact( "运行标志位" )
      Contact( "模式切换".入库模式.中间 )
      Contact( "模式切换".出库模式.全部出库完成 )
      P_Trig( "模式切换".沿."2" )
      wire#w12
      S_Coil( "模式切换".入库模式.启动 )
   END_RUNG
   RUNG wire#w12
      R_Coil( "模式切换".出库模式.启动 )
   END_RUNG
   RUNG wire#w12
      R_Coil( "模式切换".入库模式.中间 )
   END_RUNG
   // the same network as SCL:
   IF "启动" AND NOT "停止中" THEN "运行标志位" := TRUE; END_IF;
   #_w1 := "停止中" AND "模式切换".出库模式.全部出库完成 AND NOT "模式切换".沿."5";   // rising edge of "模式切换".出库模式.全部出库完成
   "模式切换".沿."5" := "模式切换".出库模式.全部出库完成;
   IF ("停止中" AND "模式切换".入库模式.入库完成保持.汇总) OR #_w1 THEN
       "运行标志位" := FALSE;
       "模式切换".入库模式.入库完成保持."1" := FALSE;
       "模式切换".入库模式.入库完成保持."2" := FALSE;
       "模式切换".入库模式.入库完成保持."3" := FALSE;
   END_IF;
   #_w2 := ("停止中" AND "模式切换".入库模式.入库完成保持.汇总) OR #_w1;
   IF #_w2 THEN
       "停止中" := FALSE;
       "模式切换".入库模式.入库完成保持."1" := FALSE;
       "模式切换".入库模式.入库完成保持."2" := FALSE;
       "模式切换".入库模式.入库完成保持."3" := FALSE;
   END_IF;
   IF "停止" THEN
       "停止中" := TRUE;
       "模式切换".入库模式.中间 := FALSE;
       "模式切换".入库模式.启动 := FALSE;
       "模式切换".出库模式.中间 := FALSE;
       "模式切换".出库模式.启动 := FALSE;
   END_IF;
   IF "运行标志位" AND "出库模式" THEN
       "模式切换".出库模式.中间 := TRUE;
       "模式切换".入库模式.中间 := FALSE;
       "模式切换".入库模式.启动 := FALSE;
   END_IF;
   #_w3 := "运行标志位" AND "模式切换".出库模式.启动 AND "1号仓库汇总块_DB".出库完成或未启用出库模式;
   "模式切换".出库模式.确认数量 := #_w3 AND "确认数量";
   IF #_w3 AND "取消" THEN
       "模式切换".出库模式.中间 := FALSE;
       "模式切换".出库模式.启动 := FALSE;
       "模式切换".入库模式.中间 := TRUE;
       "取消" := FALSE;
   END_IF;
   #_w4 := "运行标志位" AND "模式切换".出库模式.中间;
   #_w5 := #_w4 AND "模式切换".入库模式.入库完成保持.汇总;
   #_w6 := #_w5 AND NOT "模式切换".沿."1";   // rising edge
   "模式切换".沿."1" := #_w5;
   IF #_w6 THEN
       "模式切换".出库模式.启动 := TRUE;
       "模式切换".入库模式.入库完成保持."1" := FALSE;
       "模式切换".入库模式.入库完成保持."2" := FALSE;
       "模式切换".入库模式.入库完成保持."3" := FALSE;
   END_IF;
   IF #_w4 AND "1号仓库汇总块_DB".满仓信号 AND "2号仓库汇总块_DB".满仓信号 AND "3号仓库汇总块_DB".满仓信号 THEN
       "模式切换".出库模式.启动 := TRUE;
   END_IF;
   #_w7 := "运行标志位" AND "模式切换".出库模式.全部出库完成 AND NOT "模式切换".沿."3";   // rising edge of "模式切换".出库模式.全部出库完成
   "模式切换".沿."3" := "模式切换".出库模式.全部出库完成;
   #_w8 := "运行标志位" AND NOT "模式切换".沿."4";   // rising edge of "运行标志位"
   "模式切换".沿."4" := "运行标志位";
   IF ("运行标志位" AND "入库模式") OR #_w7 OR ("运行标志位" AND "取消") OR #_w8 THEN
       "模式切换".入库模式.中间 := TRUE;
       "模式切换".出库模式.中间 := FALSE;
   END_IF;
   #_w9 := "运行标志位" AND "模式切换".入库模式.中间 AND "模式切换".出库模式.全部出库完成;
   #_w10 := #_w9 AND NOT "模式切换".沿."2";   // rising edge
   "模式切换".沿."2" := #_w9;
   IF #_w10 THEN
       "模式切换".入库模式.启动 := TRUE;
       "模式切换".出库模式.启动 := FALSE;
       "模式切换".入库模式.中间 := FALSE;
   END_IF;
END_REGION

REGION Network 4
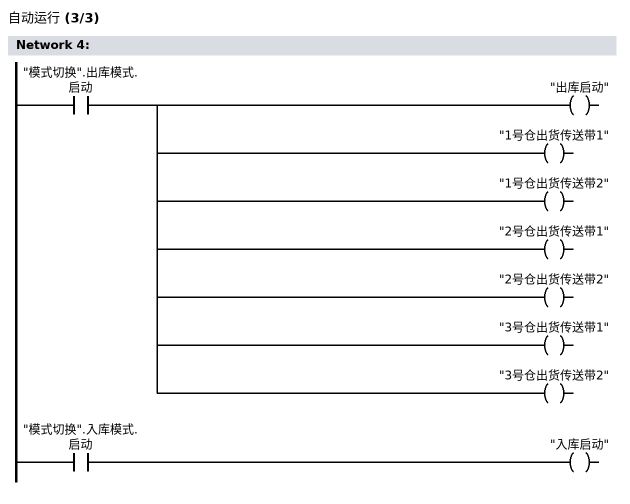
   RUNG wire#powerrail
      Contact( "模式切换".出库模式.启动 )
      wire#w1
      Coil( "出库启动" )
   END_RUNG
   RUNG wire#w1
      Coil( "1号仓出货传送带1" )
   END_RUNG
   RUNG wire#w1
      Coil( "1号仓出货传送带2" )
   END_RUNG
   RUNG wire#w1
      Coil( "2号仓出货传送带1" )
   END_RUNG
   RUNG wire#w1
      Coil( "2号仓出货传送带2" )
   END_RUNG
   RUNG wire#w1
      Coil( "3号仓出货传送带1" )
   END_RUNG
   RUNG wire#w1
      Coil( "3号仓出货传送带2" )
   END_RUNG
   RUNG wire#powerrail
      Contact( "模式切换".入库模式.启动 )
      Coil( "入库启动" )
   END_RUNG
   // the same network as SCL:
   "出库启动" := "模式切换".出库模式.启动;
   "1号仓出货传送带1" := "模式切换".出库模式.启动;
   "1号仓出货传送带2" := "模式切换".出库模式.启动;
   "2号仓出货传送带1" := "模式切换".出库模式.启动;
   "2号仓出货传送带2" := "模式切换".出库模式.启动;
   "3号仓出货传送带1" := "模式切换".出库模式.启动;
   "3号仓出货传送带2" := "模式切换".出库模式.启动;
   "入库启动" := "模式切换".入库模式.启动;
END_REGION
END_FUNCTION

FUNCTION "手动调试" : Void   // FC2, LAD
{ S7_Optimized_Access := 'TRUE' }
VERSION : 0.1
BEGIN

REGION Network 1: 传感器
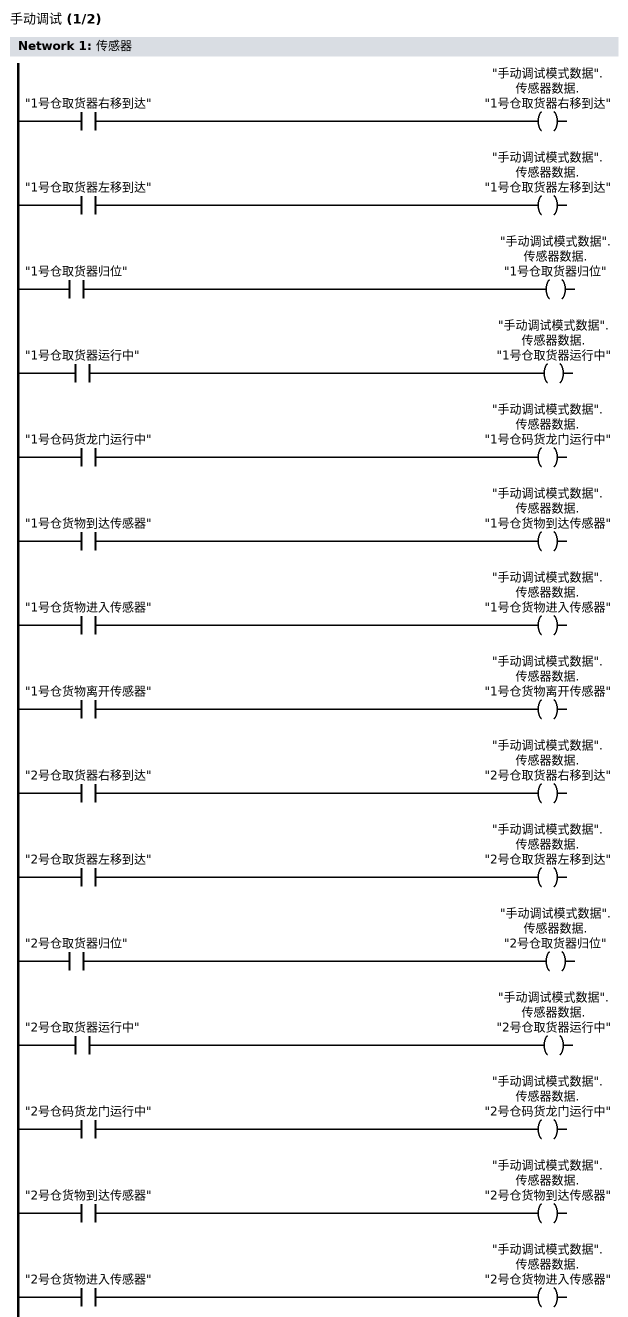
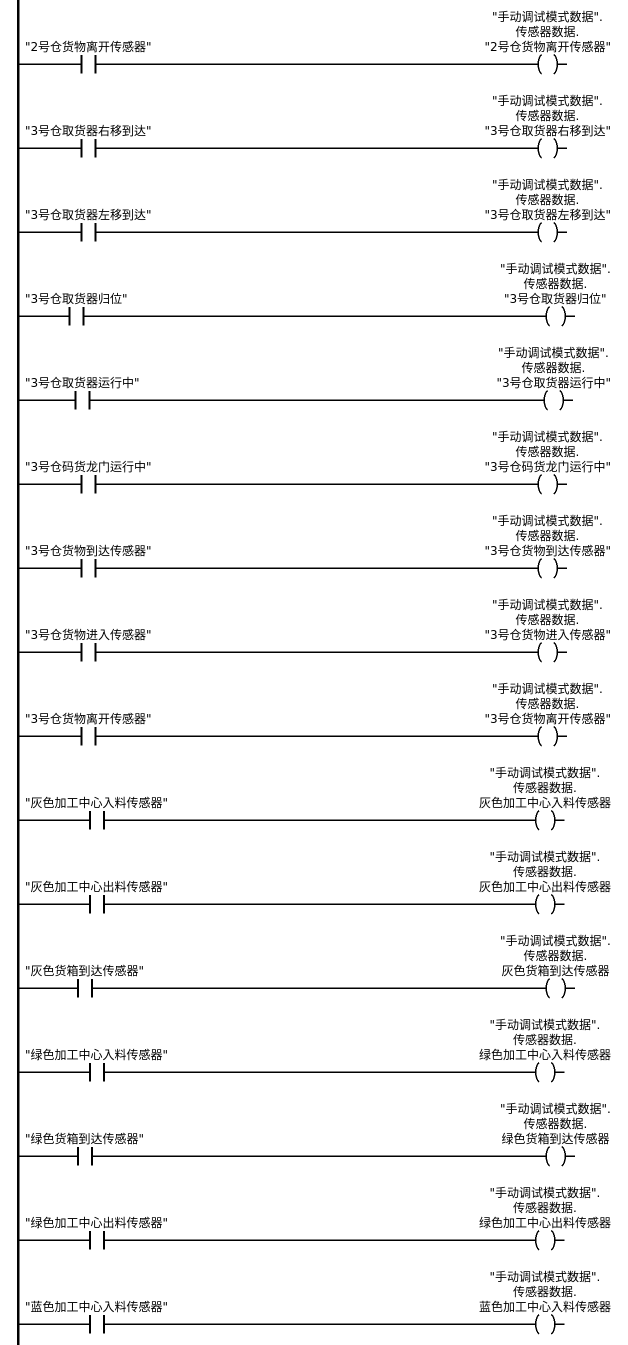
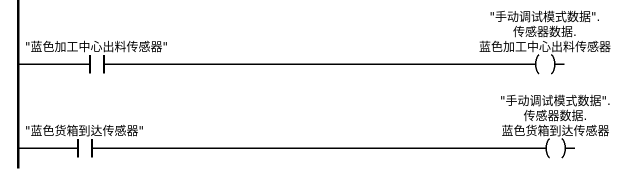
   RUNG wire#powerrail
      Contact( "1号仓取货器右移到达" )
      Coil( "手动调试模式数据".传感器数据."1号仓取货器右移到达" )
   END_RUNG
   RUNG wire#powerrail
      Contact( "1号仓取货器左移到达" )
      Coil( "手动调试模式数据".传感器数据."1号仓取货器左移到达" )
   END_RUNG
   RUNG wire#powerrail
      Contact( "1号仓取货器归位" )
      Coil( "手动调试模式数据".传感器数据."1号仓取货器归位" )
   END_RUNG
   RUNG wire#powerrail
      Contact( "1号仓取货器运行中" )
      Coil( "手动调试模式数据".传感器数据."1号仓取货器运行中" )
   END_RUNG
   RUNG wire#powerrail
      Contact( "1号仓码货龙门运行中" )
      Coil( "手动调试模式数据".传感器数据."1号仓码货龙门运行中" )
   END_RUNG
   RUNG wire#powerrail
      Contact( "1号仓货物到达传感器" )
      Coil( "手动调试模式数据".传感器数据."1号仓货物到达传感器" )
   END_RUNG
   RUNG wire#powerrail
      Contact( "1号仓货物进入传感器" )
      Coil( "手动调试模式数据".传感器数据."1号仓货物进入传感器" )
   END_RUNG
   RUNG wire#powerrail
      Contact( "1号仓货物离开传感器" )
      Coil( "手动调试模式数据".传感器数据."1号仓货物离开传感器" )
   END_RUNG
   RUNG wire#powerrail
      Contact( "2号仓取货器右移到达" )
      Coil( "手动调试模式数据".传感器数据."2号仓取货器右移到达" )
   END_RUNG
   RUNG wire#powerrail
      Contact( "2号仓取货器左移到达" )
      Coil( "手动调试模式数据".传感器数据."2号仓取货器左移到达" )
   END_RUNG
   RUNG wire#powerrail
      Contact( "2号仓取货器归位" )
      Coil( "手动调试模式数据".传感器数据."2号仓取货器归位" )
   END_RUNG
   RUNG wire#powerrail
      Contact( "2号仓取货器运行中" )
      Coil( "手动调试模式数据".传感器数据."2号仓取货器运行中" )
   END_RUNG
   RUNG wire#powerrail
      Contact( "2号仓码货龙门运行中" )
      Coil( "手动调试模式数据".传感器数据."2号仓码货龙门运行中" )
   END_RUNG
   RUNG wire#powerrail
      Contact( "2号仓货物到达传感器" )
      Coil( "手动调试模式数据".传感器数据."2号仓货物到达传感器" )
   END_RUNG
   RUNG wire#powerrail
      Contact( "2号仓货物进入传感器" )
      Coil( "手动调试模式数据".传感器数据."2号仓货物进入传感器" )
   END_RUNG
   RUNG wire#powerrail
      Contact( "2号仓货物离开传感器" )
      Coil( "手动调试模式数据".传感器数据."2号仓货物离开传感器" )
   END_RUNG
   RUNG wire#powerrail
      Contact( "3号仓取货器右移到达" )
      Coil( "手动调试模式数据".传感器数据."3号仓取货器右移到达" )
   END_RUNG
   RUNG wire#powerrail
      Contact( "3号仓取货器左移到达" )
      Coil( "手动调试模式数据".传感器数据."3号仓取货器左移到达" )
   END_RUNG
   RUNG wire#powerrail
      Contact( "3号仓取货器归位" )
      Coil( "手动调试模式数据".传感器数据."3号仓取货器归位" )
   END_RUNG
   RUNG wire#powerrail
      Contact( "3号仓取货器运行中" )
      Coil( "手动调试模式数据".传感器数据."3号仓取货器运行中" )
   END_RUNG
   RUNG wire#powerrail
      Contact( "3号仓码货龙门运行中" )
      Coil( "手动调试模式数据".传感器数据."3号仓码货龙门运行中" )
   END_RUNG
   RUNG wire#powerrail
      Contact( "3号仓货物到达传感器" )
      Coil( "手动调试模式数据".传感器数据."3号仓货物到达传感器" )
   END_RUNG
   RUNG wire#powerrail
      Contact( "3号仓货物进入传感器" )
      Coil( "手动调试模式数据".传感器数据."3号仓货物进入传感器" )
   END_RUNG
   RUNG wire#powerrail
      Contact( "3号仓货物离开传感器" )
      Coil( "手动调试模式数据".传感器数据."3号仓货物离开传感器" )
   END_RUNG
   RUNG wire#powerrail
      Contact( "灰色加工中心入料传感器" )
      Coil( "手动调试模式数据".传感器数据.灰色加工中心入料传感器 )
   END_RUNG
   RUNG wire#powerrail
      Contact( "灰色加工中心出料传感器" )
      Coil( "手动调试模式数据".传感器数据.灰色加工中心出料传感器 )
   END_RUNG
   RUNG wire#powerrail
      Contact( "灰色货箱到达传感器" )
      Coil( "手动调试模式数据".传感器数据.灰色货箱到达传感器 )
   END_RUNG
   RUNG wire#powerrail
      Contact( "绿色加工中心入料传感器" )
      Coil( "手动调试模式数据".传感器数据.绿色加工中心入料传感器 )
   END_RUNG
   RUNG wire#powerrail
      Contact( "绿色货箱到达传感器" )
      Coil( "手动调试模式数据".传感器数据.绿色货箱到达传感器 )
   END_RUNG
   RUNG wire#powerrail
      Contact( "绿色加工中心出料传感器" )
      Coil( "手动调试模式数据".传感器数据.绿色加工中心出料传感器 )
   END_RUNG
   RUNG wire#powerrail
      Contact( "蓝色加工中心入料传感器" )
      Coil( "手动调试模式数据".传感器数据.蓝色加工中心入料传感器 )
   END_RUNG
   RUNG wire#powerrail
      Contact( "蓝色加工中心出料传感器" )
      Coil( "手动调试模式数据".传感器数据.蓝色加工中心出料传感器 )
   END_RUNG
   RUNG wire#powerrail
      Contact( "蓝色货箱到达传感器" )
      Coil( "手动调试模式数据".传感器数据.蓝色货箱到达传感器 )
   END_RUNG
   // the same network as SCL:
   "手动调试模式数据".传感器数据."1号仓取货器右移到达" := "1号仓取货器右移到达";
   "手动调试模式数据".传感器数据."1号仓取货器左移到达" := "1号仓取货器左移到达";
   "手动调试模式数据".传感器数据."1号仓取货器归位" := "1号仓取货器归位";
   "手动调试模式数据".传感器数据."1号仓取货器运行中" := "1号仓取货器运行中";
   "手动调试模式数据".传感器数据."1号仓码货龙门运行中" := "1号仓码货龙门运行中";
   "手动调试模式数据".传感器数据."1号仓货物到达传感器" := "1号仓货物到达传感器";
   "手动调试模式数据".传感器数据."1号仓货物进入传感器" := "1号仓货物进入传感器";
   "手动调试模式数据".传感器数据."1号仓货物离开传感器" := "1号仓货物离开传感器";
   "手动调试模式数据".传感器数据."2号仓取货器右移到达" := "2号仓取货器右移到达";
   "手动调试模式数据".传感器数据."2号仓取货器左移到达" := "2号仓取货器左移到达";
   "手动调试模式数据".传感器数据."2号仓取货器归位" := "2号仓取货器归位";
   "手动调试模式数据".传感器数据."2号仓取货器运行中" := "2号仓取货器运行中";
   "手动调试模式数据".传感器数据."2号仓码货龙门运行中" := "2号仓码货龙门运行中";
   "手动调试模式数据".传感器数据."2号仓货物到达传感器" := "2号仓货物到达传感器";
   "手动调试模式数据".传感器数据."2号仓货物进入传感器" := "2号仓货物进入传感器";
   "手动调试模式数据".传感器数据."2号仓货物离开传感器" := "2号仓货物离开传感器";
   "手动调试模式数据".传感器数据."3号仓取货器右移到达" := "3号仓取货器右移到达";
   "手动调试模式数据".传感器数据."3号仓取货器左移到达" := "3号仓取货器左移到达";
   "手动调试模式数据".传感器数据."3号仓取货器归位" := "3号仓取货器归位";
   "手动调试模式数据".传感器数据."3号仓取货器运行中" := "3号仓取货器运行中";
   "手动调试模式数据".传感器数据."3号仓码货龙门运行中" := "3号仓码货龙门运行中";
   "手动调试模式数据".传感器数据."3号仓货物到达传感器" := "3号仓货物到达传感器";
   "手动调试模式数据".传感器数据."3号仓货物进入传感器" := "3号仓货物进入传感器";
   "手动调试模式数据".传感器数据."3号仓货物离开传感器" := "3号仓货物离开传感器";
   "手动调试模式数据".传感器数据.灰色加工中心入料传感器 := "灰色加工中心入料传感器";
   "手动调试模式数据".传感器数据.灰色加工中心出料传感器 := "灰色加工中心出料传感器";
   "手动调试模式数据".传感器数据.灰色货箱到达传感器 := "灰色货箱到达传感器";
   "手动调试模式数据".传感器数据.绿色加工中心入料传感器 := "绿色加工中心入料传感器";
   "手动调试模式数据".传感器数据.绿色货箱到达传感器 := "绿色货箱到达传感器";
   "手动调试模式数据".传感器数据.绿色加工中心出料传感器 := "绿色加工中心出料传感器";
   "手动调试模式数据".传感器数据.蓝色加工中心入料传感器 := "蓝色加工中心入料传感器";
   "手动调试模式数据".传感器数据.蓝色加工中心出料传感器 := "蓝色加工中心出料传感器";
   "手动调试模式数据".传感器数据.蓝色货箱到达传感器 := "蓝色货箱到达传感器";
END_REGION

REGION Network 2
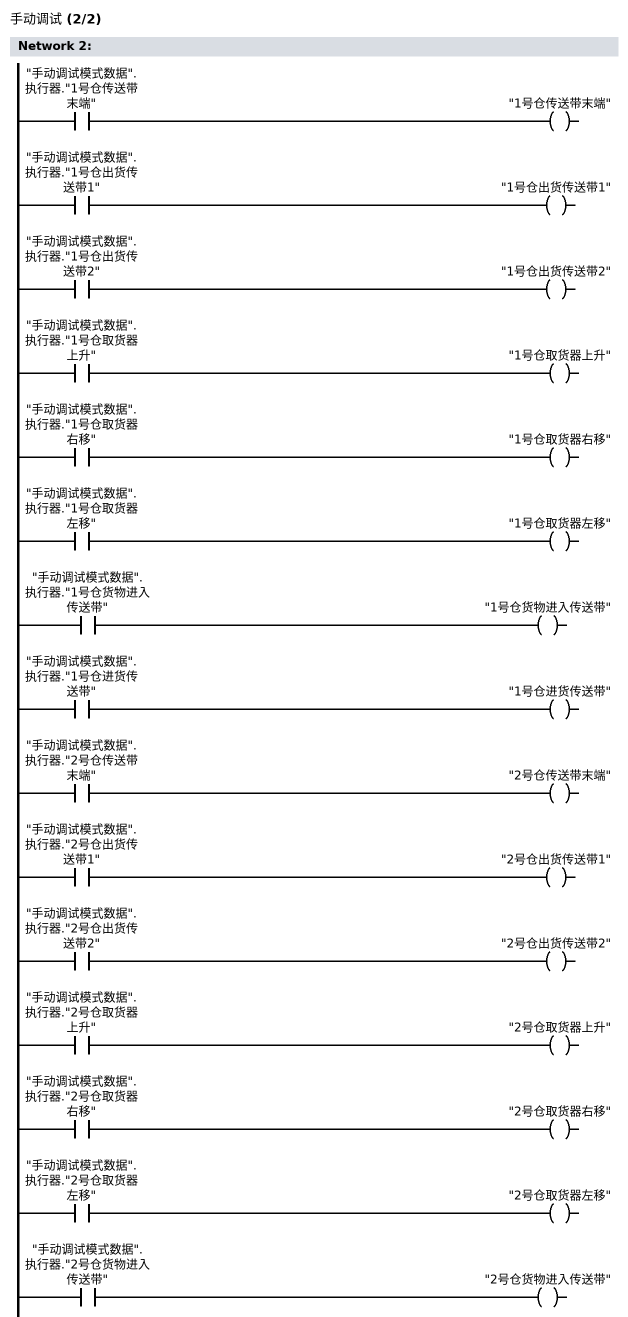
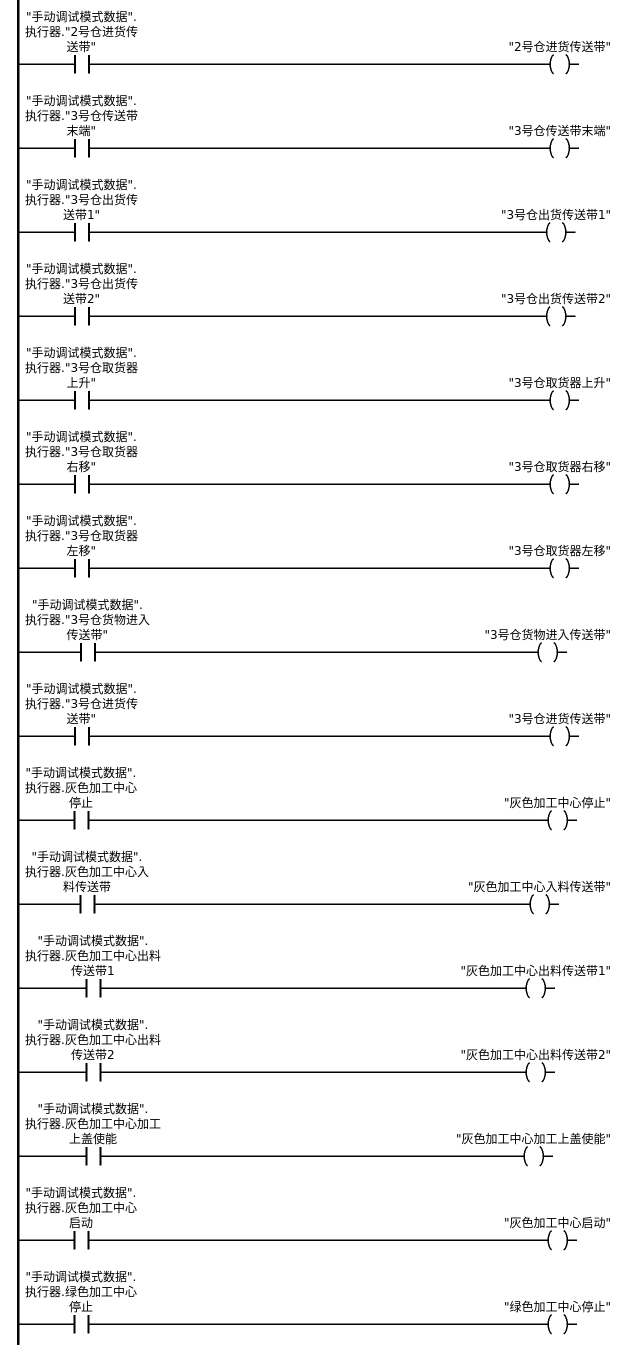
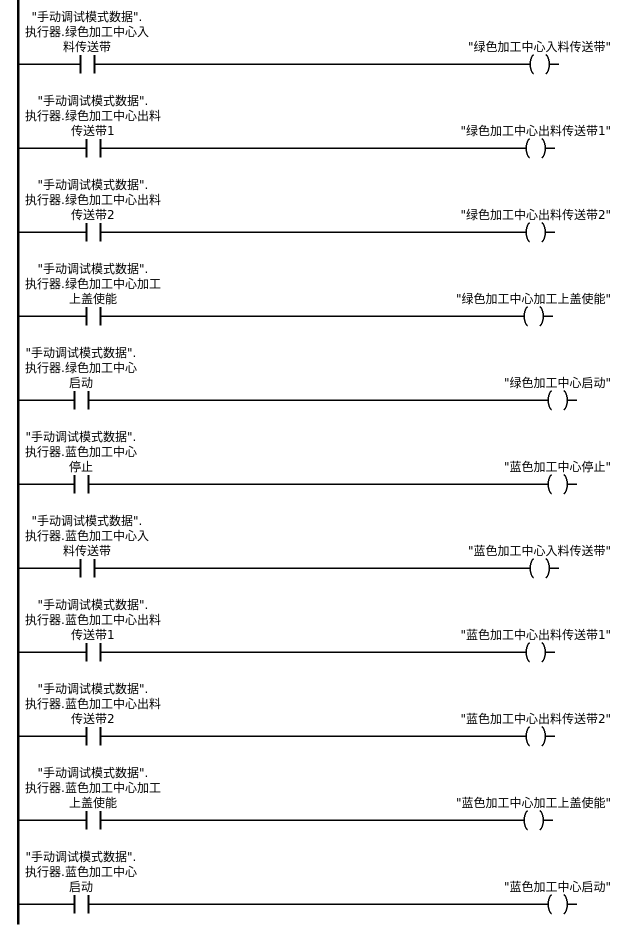
   RUNG wire#powerrail
      Contact( "手动调试模式数据".执行器."1号仓传送带末端" )
      Coil( "1号仓传送带末端" )
   END_RUNG
   RUNG wire#powerrail
      Contact( "手动调试模式数据".执行器."1号仓出货传送带1" )
      Coil( "1号仓出货传送带1" )
   END_RUNG
   RUNG wire#powerrail
      Contact( "手动调试模式数据".执行器."1号仓出货传送带2" )
      Coil( "1号仓出货传送带2" )
   END_RUNG
   RUNG wire#powerrail
      Contact( "手动调试模式数据".执行器."1号仓取货器上升" )
      Coil( "1号仓取货器上升" )
   END_RUNG
   RUNG wire#powerrail
      Contact( "手动调试模式数据".执行器."1号仓取货器右移" )
      Coil( "1号仓取货器右移" )
   END_RUNG
   RUNG wire#powerrail
      Contact( "手动调试模式数据".执行器."1号仓取货器左移" )
      Coil( "1号仓取货器左移" )
   END_RUNG
   RUNG wire#powerrail
      Contact( "手动调试模式数据".执行器."1号仓货物进入传送带" )
      Coil( "1号仓货物进入传送带" )
   END_RUNG
   RUNG wire#powerrail
      Contact( "手动调试模式数据".执行器."1号仓进货传送带" )
      Coil( "1号仓进货传送带" )
   END_RUNG
   RUNG wire#powerrail
      Contact( "手动调试模式数据".执行器."2号仓传送带末端" )
      Coil( "2号仓传送带末端" )
   END_RUNG
   RUNG wire#powerrail
      Contact( "手动调试模式数据".执行器."2号仓出货传送带1" )
      Coil( "2号仓出货传送带1" )
   END_RUNG
   RUNG wire#powerrail
      Contact( "手动调试模式数据".执行器."2号仓出货传送带2" )
      Coil( "2号仓出货传送带2" )
   END_RUNG
   RUNG wire#powerrail
      Contact( "手动调试模式数据".执行器."2号仓取货器上升" )
      Coil( "2号仓取货器上升" )
   END_RUNG
   RUNG wire#powerrail
      Contact( "手动调试模式数据".执行器."2号仓取货器右移" )
      Coil( "2号仓取货器右移" )
   END_RUNG
   RUNG wire#powerrail
      Contact( "手动调试模式数据".执行器."2号仓取货器左移" )
      Coil( "2号仓取货器左移" )
   END_RUNG
   RUNG wire#powerrail
      Contact( "手动调试模式数据".执行器."2号仓货物进入传送带" )
      Coil( "2号仓货物进入传送带" )
   END_RUNG
   RUNG wire#powerrail
      Contact( "手动调试模式数据".执行器."2号仓进货传送带" )
      Coil( "2号仓进货传送带" )
   END_RUNG
   RUNG wire#powerrail
      Contact( "手动调试模式数据".执行器."3号仓传送带末端" )
      Coil( "3号仓传送带末端" )
   END_RUNG
   RUNG wire#powerrail
      Contact( "手动调试模式数据".执行器."3号仓出货传送带1" )
      Coil( "3号仓出货传送带1" )
   END_RUNG
   RUNG wire#powerrail
      Contact( "手动调试模式数据".执行器."3号仓出货传送带2" )
      Coil( "3号仓出货传送带2" )
   END_RUNG
   RUNG wire#powerrail
      Contact( "手动调试模式数据".执行器."3号仓取货器上升" )
      Coil( "3号仓取货器上升" )
   END_RUNG
   RUNG wire#powerrail
      Contact( "手动调试模式数据".执行器."3号仓取货器右移" )
      Coil( "3号仓取货器右移" )
   END_RUNG
   RUNG wire#powerrail
      Contact( "手动调试模式数据".执行器."3号仓取货器左移" )
      Coil( "3号仓取货器左移" )
   END_RUNG
   RUNG wire#powerrail
      Contact( "手动调试模式数据".执行器."3号仓货物进入传送带" )
      Coil( "3号仓货物进入传送带" )
   END_RUNG
   RUNG wire#powerrail
      Contact( "手动调试模式数据".执行器."3号仓进货传送带" )
      Coil( "3号仓进货传送带" )
   END_RUNG
   RUNG wire#powerrail
      Contact( "手动调试模式数据".执行器.灰色加工中心停止 )
      Coil( "灰色加工中心停止" )
   END_RUNG
   RUNG wire#powerrail
      Contact( "手动调试模式数据".执行器.灰色加工中心入料传送带 )
      Coil( "灰色加工中心入料传送带" )
   END_RUNG
   RUNG wire#powerrail
      Contact( "手动调试模式数据".执行器.灰色加工中心出料传送带1 )
      Coil( "灰色加工中心出料传送带1" )
   END_RUNG
   RUNG wire#powerrail
      Contact( "手动调试模式数据".执行器.灰色加工中心出料传送带2 )
      Coil( "灰色加工中心出料传送带2" )
   END_RUNG
   RUNG wire#powerrail
      Contact( "手动调试模式数据".执行器.灰色加工中心加工上盖使能 )
      Coil( "灰色加工中心加工上盖使能" )
   END_RUNG
   RUNG wire#powerrail
      Contact( "手动调试模式数据".执行器.灰色加工中心启动 )
      Coil( "灰色加工中心启动" )
   END_RUNG
   RUNG wire#powerrail
      Contact( "手动调试模式数据".执行器.绿色加工中心停止 )
      Coil( "绿色加工中心停止" )
   END_RUNG
   RUNG wire#powerrail
      Contact( "手动调试模式数据".执行器.绿色加工中心入料传送带 )
      Coil( "绿色加工中心入料传送带" )
   END_RUNG
   RUNG wire#powerrail
      Contact( "手动调试模式数据".执行器.绿色加工中心出料传送带1 )
      Coil( "绿色加工中心出料传送带1" )
   END_RUNG
   RUNG wire#powerrail
      Contact( "手动调试模式数据".执行器.绿色加工中心出料传送带2 )
      Coil( "绿色加工中心出料传送带2" )
   END_RUNG
   RUNG wire#powerrail
      Contact( "手动调试模式数据".执行器.绿色加工中心加工上盖使能 )
      Coil( "绿色加工中心加工上盖使能" )
   END_RUNG
   RUNG wire#powerrail
      Contact( "手动调试模式数据".执行器.绿色加工中心启动 )
      Coil( "绿色加工中心启动" )
   END_RUNG
   RUNG wire#powerrail
      Contact( "手动调试模式数据".执行器.蓝色加工中心停止 )
      Coil( "蓝色加工中心停止" )
   END_RUNG
   RUNG wire#powerrail
      Contact( "手动调试模式数据".执行器.蓝色加工中心入料传送带 )
      Coil( "蓝色加工中心入料传送带" )
   END_RUNG
   RUNG wire#powerrail
      Contact( "手动调试模式数据".执行器.蓝色加工中心出料传送带1 )
      Coil( "蓝色加工中心出料传送带1" )
   END_RUNG
   RUNG wire#powerrail
      Contact( "手动调试模式数据".执行器.蓝色加工中心出料传送带2 )
      Coil( "蓝色加工中心出料传送带2" )
   END_RUNG
   RUNG wire#powerrail
      Contact( "手动调试模式数据".执行器.蓝色加工中心加工上盖使能 )
      Coil( "蓝色加工中心加工上盖使能" )
   END_RUNG
   RUNG wire#powerrail
      Contact( "手动调试模式数据".执行器.蓝色加工中心启动 )
      Coil( "蓝色加工中心启动" )
   END_RUNG
   // the same network as SCL:
   "1号仓传送带末端" := "手动调试模式数据".执行器."1号仓传送带末端";
   "1号仓出货传送带1" := "手动调试模式数据".执行器."1号仓出货传送带1";
   "1号仓出货传送带2" := "手动调试模式数据".执行器."1号仓出货传送带2";
   "1号仓取货器上升" := "手动调试模式数据".执行器."1号仓取货器上升";
   "1号仓取货器右移" := "手动调试模式数据".执行器."1号仓取货器右移";
   "1号仓取货器左移" := "手动调试模式数据".执行器."1号仓取货器左移";
   "1号仓货物进入传送带" := "手动调试模式数据".执行器."1号仓货物进入传送带";
   "1号仓进货传送带" := "手动调试模式数据".执行器."1号仓进货传送带";
   "2号仓传送带末端" := "手动调试模式数据".执行器."2号仓传送带末端";
   "2号仓出货传送带1" := "手动调试模式数据".执行器."2号仓出货传送带1";
   "2号仓出货传送带2" := "手动调试模式数据".执行器."2号仓出货传送带2";
   "2号仓取货器上升" := "手动调试模式数据".执行器."2号仓取货器上升";
   "2号仓取货器右移" := "手动调试模式数据".执行器."2号仓取货器右移";
   "2号仓取货器左移" := "手动调试模式数据".执行器."2号仓取货器左移";
   "2号仓货物进入传送带" := "手动调试模式数据".执行器."2号仓货物进入传送带";
   "2号仓进货传送带" := "手动调试模式数据".执行器."2号仓进货传送带";
   "3号仓传送带末端" := "手动调试模式数据".执行器."3号仓传送带末端";
   "3号仓出货传送带1" := "手动调试模式数据".执行器."3号仓出货传送带1";
   "3号仓出货传送带2" := "手动调试模式数据".执行器."3号仓出货传送带2";
   "3号仓取货器上升" := "手动调试模式数据".执行器."3号仓取货器上升";
   "3号仓取货器右移" := "手动调试模式数据".执行器."3号仓取货器右移";
   "3号仓取货器左移" := "手动调试模式数据".执行器."3号仓取货器左移";
   "3号仓货物进入传送带" := "手动调试模式数据".执行器."3号仓货物进入传送带";
   "3号仓进货传送带" := "手动调试模式数据".执行器."3号仓进货传送带";
   "灰色加工中心停止" := "手动调试模式数据".执行器.灰色加工中心停止;
   "灰色加工中心入料传送带" := "手动调试模式数据".执行器.灰色加工中心入料传送带;
   "灰色加工中心出料传送带1" := "手动调试模式数据".执行器.灰色加工中心出料传送带1;
   "灰色加工中心出料传送带2" := "手动调试模式数据".执行器.灰色加工中心出料传送带2;
   "灰色加工中心加工上盖使能" := "手动调试模式数据".执行器.灰色加工中心加工上盖使能;
   "灰色加工中心启动" := "手动调试模式数据".执行器.灰色加工中心启动;
   "绿色加工中心停止" := "手动调试模式数据".执行器.绿色加工中心停止;
   "绿色加工中心入料传送带" := "手动调试模式数据".执行器.绿色加工中心入料传送带;
   "绿色加工中心出料传送带1" := "手动调试模式数据".执行器.绿色加工中心出料传送带1;
   "绿色加工中心出料传送带2" := "手动调试模式数据".执行器.绿色加工中心出料传送带2;
   "绿色加工中心加工上盖使能" := "手动调试模式数据".执行器.绿色加工中心加工上盖使能;
   "绿色加工中心启动" := "手动调试模式数据".执行器.绿色加工中心启动;
   "蓝色加工中心停止" := "手动调试模式数据".执行器.蓝色加工中心停止;
   "蓝色加工中心入料传送带" := "手动调试模式数据".执行器.蓝色加工中心入料传送带;
   "蓝色加工中心出料传送带1" := "手动调试模式数据".执行器.蓝色加工中心出料传送带1;
   "蓝色加工中心出料传送带2" := "手动调试模式数据".执行器.蓝色加工中心出料传送带2;
   "蓝色加工中心加工上盖使能" := "手动调试模式数据".执行器.蓝色加工中心加工上盖使能;
   "蓝色加工中心启动" := "手动调试模式数据".执行器.蓝色加工中心启动;
END_REGION
END_FUNCTION

FUNCTION "急停" : Void   // FC3, LAD
{ S7_Optimized_Access := 'TRUE' }
VERSION : 0.1
BEGIN

REGION Network 1
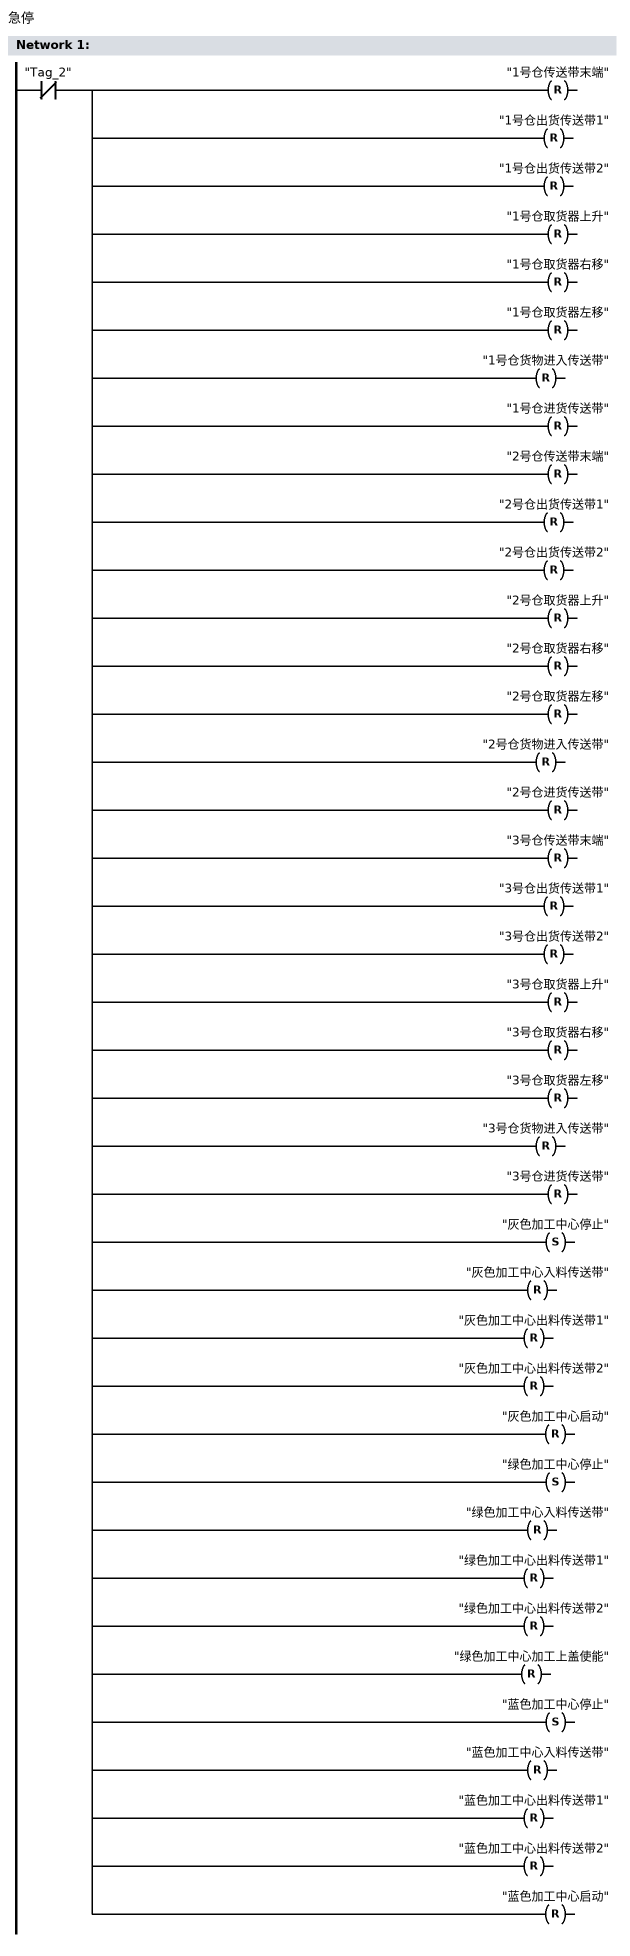
   RUNG wire#powerrail
      I_Contact( "Tag_2" )
      wire#w1
      R_Coil( "1号仓传送带末端" )
   END_RUNG
   RUNG wire#w1
      R_Coil( "1号仓出货传送带1" )
   END_RUNG
   RUNG wire#w1
      R_Coil( "1号仓出货传送带2" )
   END_RUNG
   RUNG wire#w1
      R_Coil( "1号仓取货器上升" )
   END_RUNG
   RUNG wire#w1
      R_Coil( "1号仓取货器右移" )
   END_RUNG
   RUNG wire#w1
      R_Coil( "1号仓取货器左移" )
   END_RUNG
   RUNG wire#w1
      R_Coil( "1号仓货物进入传送带" )
   END_RUNG
   RUNG wire#w1
      R_Coil( "1号仓进货传送带" )
   END_RUNG
   RUNG wire#w1
      R_Coil( "2号仓传送带末端" )
   END_RUNG
   RUNG wire#w1
      R_Coil( "2号仓出货传送带1" )
   END_RUNG
   RUNG wire#w1
      R_Coil( "2号仓出货传送带2" )
   END_RUNG
   RUNG wire#w1
      R_Coil( "2号仓取货器上升" )
   END_RUNG
   RUNG wire#w1
      R_Coil( "2号仓取货器右移" )
   END_RUNG
   RUNG wire#w1
      R_Coil( "2号仓取货器左移" )
   END_RUNG
   RUNG wire#w1
      R_Coil( "2号仓货物进入传送带" )
   END_RUNG
   RUNG wire#w1
      R_Coil( "2号仓进货传送带" )
   END_RUNG
   RUNG wire#w1
      R_Coil( "3号仓传送带末端" )
   END_RUNG
   RUNG wire#w1
      R_Coil( "3号仓出货传送带1" )
   END_RUNG
   RUNG wire#w1
      R_Coil( "3号仓出货传送带2" )
   END_RUNG
   RUNG wire#w1
      R_Coil( "3号仓取货器上升" )
   END_RUNG
   RUNG wire#w1
      R_Coil( "3号仓取货器右移" )
   END_RUNG
   RUNG wire#w1
      R_Coil( "3号仓取货器左移" )
   END_RUNG
   RUNG wire#w1
      R_Coil( "3号仓货物进入传送带" )
   END_RUNG
   RUNG wire#w1
      R_Coil( "3号仓进货传送带" )
   END_RUNG
   RUNG wire#w1
      S_Coil( "灰色加工中心停止" )
   END_RUNG
   RUNG wire#w1
      R_Coil( "灰色加工中心入料传送带" )
   END_RUNG
   RUNG wire#w1
      R_Coil( "灰色加工中心出料传送带1" )
   END_RUNG
   RUNG wire#w1
      R_Coil( "灰色加工中心出料传送带2" )
   END_RUNG
   RUNG wire#w1
      R_Coil( "灰色加工中心启动" )
   END_RUNG
   RUNG wire#w1
      S_Coil( "绿色加工中心停止" )
   END_RUNG
   RUNG wire#w1
      R_Coil( "绿色加工中心入料传送带" )
   END_RUNG
   RUNG wire#w1
      R_Coil( "绿色加工中心出料传送带1" )
   END_RUNG
   RUNG wire#w1
      R_Coil( "绿色加工中心出料传送带2" )
   END_RUNG
   RUNG wire#w1
      R_Coil( "绿色加工中心加工上盖使能" )
   END_RUNG
   RUNG wire#w1
      S_Coil( "蓝色加工中心停止" )
   END_RUNG
   RUNG wire#w1
      R_Coil( "蓝色加工中心入料传送带" )
   END_RUNG
   RUNG wire#w1
      R_Coil( "蓝色加工中心出料传送带1" )
   END_RUNG
   RUNG wire#w1
      R_Coil( "蓝色加工中心出料传送带2" )
   END_RUNG
   RUNG wire#w1
      R_Coil( "蓝色加工中心启动" )
   END_RUNG
   // the same network as SCL:
   IF NOT "Tag_2" THEN
       "1号仓传送带末端" := FALSE;
       "1号仓出货传送带1" := FALSE;
       "1号仓出货传送带2" := FALSE;
       "1号仓取货器上升" := FALSE;
       "1号仓取货器右移" := FALSE;
       "1号仓取货器左移" := FALSE;
       "1号仓货物进入传送带" := FALSE;
       "1号仓进货传送带" := FALSE;
       "2号仓传送带末端" := FALSE;
       "2号仓出货传送带1" := FALSE;
       "2号仓出货传送带2" := FALSE;
       "2号仓取货器上升" := FALSE;
       "2号仓取货器右移" := FALSE;
       "2号仓取货器左移" := FALSE;
       "2号仓货物进入传送带" := FALSE;
       "2号仓进货传送带" := FALSE;
       "3号仓传送带末端" := FALSE;
       "3号仓出货传送带1" := FALSE;
       "3号仓出货传送带2" := FALSE;
       "3号仓取货器上升" := FALSE;
       "3号仓取货器右移" := FALSE;
       "3号仓取货器左移" := FALSE;
       "3号仓货物进入传送带" := FALSE;
       "3号仓进货传送带" := FALSE;
       "灰色加工中心停止" := TRUE;
       "灰色加工中心入料传送带" := FALSE;
       "灰色加工中心出料传送带1" := FALSE;
       "灰色加工中心出料传送带2" := FALSE;
       "灰色加工中心启动" := FALSE;
       "绿色加工中心停止" := TRUE;
       "绿色加工中心入料传送带" := FALSE;
       "绿色加工中心出料传送带1" := FALSE;
       "绿色加工中心出料传送带2" := FALSE;
       "绿色加工中心加工上盖使能" := FALSE;
       "蓝色加工中心停止" := TRUE;
       "蓝色加工中心入料传送带" := FALSE;
       "蓝色加工中心出料传送带1" := FALSE;
       "蓝色加工中心出料传送带2" := FALSE;
       "蓝色加工中心启动" := FALSE;
   END_IF;
END_REGION
END_FUNCTION

FUNCTION "MHJ-PLC-Lab-Function-S71500" : Void   // FC9000, SCL
{ S7_Optimized_Access := 'TRUE' }
VERSION : 0.1
   VAR_TEMP
      Value : Byte;
      ForCounter : Int;
   END_VAR
   VAR CONSTANT
      Value_01_DW : DWord := 16#1223_5486;
      Value_02_DW : DWord := 16#A6C9_D1F5;
   END_VAR
BEGIN

   #Value:=PEEK(area := 16#82,
        dbNumber := 0,
        byteOffset := 511);
   #Value := #Value + 1;

   POKE(area := 16#82,
        dbNumber := 0,
        byteOffset := 511,
        value := #Value);

   POKE(area := 16#82,
        dbNumber := 0,
        byteOffset := 1016,
        value := #Value_01_DW);
   POKE(area := 16#82,
        dbNumber := 0,
        byteOffset := 1020,
        value := #Value_02_DW);

   FOR #ForCounter := 0 TO 63 DO
       #Value:=PEEK(area := 16#1,
            dbNumber := 0,
            byteOffset := #ForCounter);
       POKE(area := 16#81,
            dbNumber := 0,
            byteOffset := #ForCounter,
            value := #Value);
   END_FOR;
   #Value := PEEK(area := 16#1,
                  dbNumber := 0,
                  byteOffset := 512);
   POKE(area := 16#82,
        dbNumber := 0,
        byteOffset := 512,
        value := #Value);
END_FUNCTION

ORGANIZATION_BLOCK "Main"   // OB1, LAD, ProgramCycle
TITLE = "Main Program Sweep (Cycle)"
{ S7_Optimized_Access := 'TRUE' }
VERSION : 0.1
   VAR_INPUT
      Initial_Call : Bool;   // Initial call of this OB
      Remanence : Bool;   // =True, if remanent data are available
   END_VAR
   VAR_TEMP   // added for the SCL form of the ladder/FBD networks
      _w1 : Bool;
   END_VAR
BEGIN

REGION Network 2
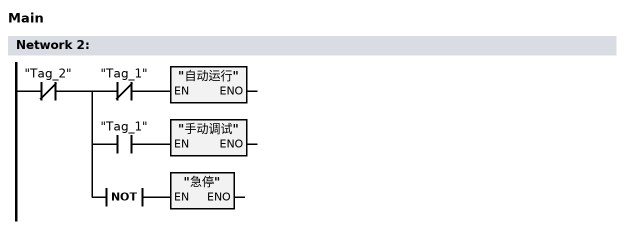
   RUNG wire#powerrail
      I_Contact( "Tag_2" )
      wire#w1
      I_Contact( "Tag_1" )
      "自动运行"()
   END_RUNG
   RUNG wire#w1
      Contact( "Tag_1" )
      "手动调试"()
   END_RUNG
   RUNG wire#w1
      Not()
      "急停"()
   END_RUNG
   // the same network as SCL:
   #_w1 := NOT "Tag_2";
   IF NOT "Tag_2" AND NOT "Tag_1" THEN "自动运行"(); END_IF;
   IF #_w1 AND "Tag_1" THEN "手动调试"(); END_IF;
   IF NOT #_w1 THEN "急停"(); END_IF;
END_REGION
END_ORGANIZATION_BLOCK